	11: IF (OP90_Camera_Trigger AND (NOT OP90_Camera_Done)) OR OP90_Miss_Trigger THEN
			OP90_LH_Camera_Trigger:=1;
			OP90_RH_Camera_Trigger:=1;
			Conv_Cam_Step		  :=15;	
		END_IF

	15:	IF LH_Cam_Completed AND RH_Cam_Completed THEN// (NOT OP90_LH_Camera_Trigger) AND (NOT OP90_RH_Camera_Trigger) THEN //(Temp_Counter_LH<OP90_Camera_FB.OP90_LH_Acquisition_ID AND Temp_Counter_RH<OP90_Camera_FB.OP90_RH_Acquisition_ID )THEN
			OP90_LH_Camera_Trigger:=0;
			OP90_RH_Camera_Trigger:=0;
			OP90_Camera_Trigger :=0;
			OP90_Miss_Trigger	:=0;
			Conv_Cam_Step:=25;
		END_IF  
	   
	25: IF OP90_Camera_FB.OP90_LH_Cam_Result[0]=1 AND OP90_Camera_FB.OP90_RH_Cam_Result[0]=1 THEN
			OP90_LH_Camera_OK:=1;
			OP90_RH_Camera_OK:=1;
			Conv_Cam_Step    :=50;
		ELSIF (OP90_Camera_FB.OP90_LH_Cam_Result[2]<>1 OR OP90_Camera_FB.OP90_RH_Cam_Result[2]<>1) THEN
			OP90_One_Cycle	 :=1;
			Comp_Not_present_Counter:=Comp_Not_present_Counter+1;
			Conv_Cam_Step    :=50;
		ELSIF (OP90_Camera_FB.OP90_LH_Cam_Result[1]=1 OR OP90_Camera_FB.OP90_RH_Cam_Result[1]=1) THEN //AND ( OP90_Camera_FB.OP90_LH_Cam_Result[2]=1 AND OP90_Camera_FB.OP90_RH_Cam_Result[2]=1) THEN			
			IF OP90_Camera_FB.OP90_LH_Cam_Result[0]=1 THEN
				OP90_LH_Camera_OK:=1;
			END_IF
			IF OP90_Camera_FB.OP90_RH_Cam_Result[0]=1 THEN
				OP90_RH_Camera_OK:=1;
			END_IF
			Conv_Cam_Step:=30;
		END_IF	
			
   30: 	IF OP90_Camera_FB.OP90_LH_Cam_Result[1]=1 THEN
	   		OP90_LH_Camera_NOK:=1;
  	    END_IF
		IF OP90_Camera_FB.OP90_RH_Cam_Result[1]=1 THEN
	   		OP90_RH_Camera_NOK:=1;
  	    END_IF
		Conv_Cam_Step:=50;
		
   50:  OP90_Camera_Done:=1;
   		Comp_Not_present_Counter:=0;
   		Temp_Counter_LH:=OP90_Camera_FB.OP90_LH_Acquisition_ID;
		Temp_Counter_RH:=OP90_Camera_FB.OP90_RH_Acquisition_ID;
		IF Camera_Trigger_Ack_OP90 THEN
			Conv_Cam_Step   :=10;
			OP90_Camera_Done:=0;
		END_IF
   	    
END_CASE

END_PROGRAM

// ---- FB/Servo_Conveyor_FB_OP90.TcPOU
FUNCTION_BLOCK Servo_Conveyor_FB_OP90
VAR_INPUT
	Conveyor_Prgrm_Start			: BOOL;
	Conveyor_Prgrm_Reset			: BOOL;
	Conveyor_Continuous_Run			: BOOL;	
	Camera_Trigger_OK				: BOOL;	
	Conveyor_Bypass					: BOOL;
	Fwd_Time_IP						: INT;
	Rev_Time_IP						: INT;
	Conveyor_FWD_Speed				: REAL;
	Conveyor_REV_Speed				: REAL;
	Conveyor_FWD_Position			: REAL;
	Conveyor_REV_Position			: REAL;	
	Velocity_mode					: BOOL;
	LH_Work_Sensor					: BOOL;
	LH_Home_Sensor					: BOOL;
	RH_Work_Sensor					: BOOL;
	RH_Home_Sensor					: BOOL;	
	LH_Camera_OK					: BOOL;
	LH_Camera_NOK					: BOOL;	
	RH_Camera_OK					: BOOL;
	RH_Camera_NOK					: BOOL;
	Track_Overflow					: BOOL;
	//Track_Sensor_FB					: BOOL;
END_VAR
VAR_OUTPUT
	Camera_Trigger_ACK				: BOOL;	
	LH_Work_Coil					: BOOL;
	LH_Home_Coil					: BOOL;
	RH_Work_Coil					: BOOL;
	RH_Home_Coil					: BOOL;	
	Ready_to_Pick					: BOOL;
	Drum_ON							: BOOL;
	Step_Num						: INT;
END_VAR
VAR_IN_OUT
	Camera_trigger						: BOOL;
	One_Cycle							: BOOL;
	Pick_Done						    : BOOL;
	Track_Sensor_FB					    : BOOL;
	Conveyor_Servo_Control_Structure	:  Servo_Control;
END_VAR
VAR
	Conveyor_Speed  : REAL;
	Cyl_Delay 		: TON;
	Cyl_Temp 		: BOOL;
	temp_3			: BOOL;
	cam_ok 			: BOOL;
	con_step_no 	: INT;	
	t1				: ton;
	t2				: ton;
	t3				: ton;
	t4				: ton;	
	count_nok   	: INT;
	forward			: BOOL;
	reverse			: BOOL;
	fwd_time		: INT;
	rev_time		: INT;
	temp            : BOOL;
	VeloCity_Frwd   : REAL := 200;
	Track_Count		: TON;
	Temp_1 : R_TRIG;
	Temp_Cont : BOOL;
	Conti_run : TON;
END_VAR

IF NOT Conveyor_Prgrm_Start OR Conveyor_Servo_Control_Structure.Axis_Error THEN
	con_step_no:=10;
	Camera_Trigger_ACK:=0;
	Ready_to_Pick:=FALSE;
	Conveyor_Servo_Control_Structure.VELmove_Start:=FALSE;
END_IF

IF Conveyor_Bypass THEN
	con_step_no:=10;
	Ready_to_Pick:=1;
	IF Pick_Done THEN
		Pick_Done:=0;
		Ready_to_Pick:=0;
	END_IF
END_IF

IF forward THEN
	Conveyor_Speed:=Conveyor_FWD_Speed;
END_IF
IF reverse THEN
	Conveyor_Speed:=Conveyor_REV_Speed;
END_IF

Conti_run(IN:=(con_step_no=25),PT:=T#2S);

CASE con_step_no OF
		10: IF Conveyor_Prgrm_Start THEN
				con_step_no:=15;
			END_IF
			
		15: LH_Home_Coil:=1;
			RH_Home_Coil:=1;	
			IF LH_Home_Sensor AND RH_Home_Sensor THEN
				LH_Home_Coil:=0;
				RH_Home_Coil:=0;
				con_step_no:= 70;
			END_IF
		
        20:	Ready_to_Pick :=FALSE;
			Pick_Done:= FALSE;
			Conveyor_Servo_Control_Structure.Velocity:= VeloCity_Frwd;		
			Conveyor_Servo_Control_Structure.VELmove_Start:=FALSE;
			IF NOT Conveyor_Servo_Control_Structure.VELmove_Start THEN
				con_step_no:= 25;
			END_IF	
			
		25:	Drum_ON:=1;
			Conveyor_Servo_Control_Structure.VELmove_Start:=TRUE;	
			IF Track_Sensor_FB THEN
				Conveyor_Servo_Control_Structure.VELmove_Start:=FALSE;
				Drum_ON	   :=FALSE;
				con_step_no:= 80;
			END_IF
	
		70: IF NOT Conveyor_Servo_Control_Structure.VELmove_Start THEN
			  Camera_trigger :=TRUE;
			  con_step_no	 := 75;
			END_IF	
					
		75:	IF Camera_Trigger_OK AND NOT Conveyor_Servo_Control_Structure.VELmove_Start AND Conveyor_Servo_Control_Structure.Axis_ready THEN
				IF LH_Camera_OK AND RH_Camera_OK THEN
				 con_step_no:= 100;
				 Camera_Trigger_ACK:=1;
				 fwd_time:=Fwd_Time_IP;
				 count_nok:=0;	
				ELSIF (LH_Camera_NOK) OR (RH_Camera_NOK) AND count_nok<5 THEN
				 count_nok := count_nok +1;
				 con_step_no:= 76;	
				ELSIF count_nok>=5 THEN
	             fwd_time:=3000;
				 con_step_no:= 80; 
				END_IF
			END_IF	
			
		76:	IF LH_Camera_NOK AND NOT Conveyor_Servo_Control_Structure.VELmove_Start THEN
				IF LH_Home_Sensor THEN
					LH_Work_Coil:=TRUE;
					Cyl_Temp:=1;
				END_IF	
				IF Cyl_Delay.Q THEN
					con_step_no:= 77;
				END_IF	
			ELSIF LH_Camera_OK AND RH_Camera_NOK THEN
				con_step_no:= 78;
			END_IF	
			
			
		77: 	IF  LH_Work_Sensor THEN
					LH_Work_Coil:=0;
					LH_Home_Coil:=1;
				END_IF	
				IF LH_Home_Sensor AND NOT LH_Work_Coil AND count_nok<5 THEN
					LH_Home_Coil:=0;
					fwd_time:=Fwd_Time_IP;
				    con_step_no:= 80;
				END_IF
                IF  LH_Home_Sensor AND NOT LH_Work_Coil AND count_nok>=5 THEN
					LH_Home_Coil:=0;
					fwd_time:=3000;
					count_nok:=0;
					//Camera_Trigger_ACK:=1;
				    con_step_no:= 80;	
				END_IF

		78:	IF RH_Camera_NOK AND NOT Conveyor_Servo_Control_Structure.VELmove_Start THEN	
				IF RH_Home_Sensor THEN
					RH_Work_Coil:=TRUE;
					Cyl_Temp:=1;
				END_IF	
				IF Cyl_Delay.Q THEN
					con_step_no:= 79;
				END_IF				
			END_IF		
			
		79: 	IF RH_Work_Sensor THEN
					RH_Work_Coil:=0;
					RH_Home_Coil:=1;				
				END_IF
				IF RH_Home_Sensor AND NOT RH_Work_Coil AND count_nok<5 THEN
					RH_Home_Coil:=0;					
					fwd_time:=Fwd_Time_IP;
				    con_step_no:= 80;
				END_IF
				IF RH_Home_Sensor AND NOT RH_Work_Coil AND count_nok>=5 THEN
					fwd_time:=3000;
					count_nok:=0;
					RH_Home_Coil:=0;
				    con_step_no:= 80;	
				END_IF
			
		80: 	IF Velocity_mode THEN
					IF fwd_time=3000 THEN
			       		count_nok:=0;	
					END_IF
                	Conveyor_Servo_Control_Structure.Velocity:= Conveyor_Speed;				
					forward:=TRUE;
					Conveyor_Servo_Control_Structure.VELmove_Start:=TRUE;	
					IF t2.Q THEN
    					forward:=FALSE;
						Conveyor_Servo_Control_Structure.VELmove_Start:=FALSE;
						Camera_Trigger_ACK:=1;
						con_step_no:= 90;
					END_IF
				ELSE
					Conveyor_Servo_Control_Structure.Velocity:=Conveyor_FWD_Speed;
					Conveyor_Servo_Control_Structure.Position:=Conveyor_FWD_Position;
					Conveyor_Servo_Control_Structure.RELmove_Start:=1;
					Camera_Trigger_ACK:=1;
					con_step_no:= 85;
				END_IF	
				
		85 : 	IF NOT Conveyor_Servo_Control_Structure.RELmove_Start THEN 
					con_step_no:= 90;
				END_IF	
		
		90: IF Velocity_mode THEN
				Conveyor_Servo_Control_Structure.Velocity:= Conveyor_Speed;
				reverse:=TRUE;
				Conveyor_Servo_Control_Structure.VELmove_Start:=TRUE;
				IF t3.Q THEN
 					reverse:=FALSE;
					Conveyor_Servo_Control_Structure.VELmove_Start:=FALSE;
					Camera_Trigger_ACK:=0;
					IF NOT Camera_Trigger_ACK THEN
						con_step_no:= 70;
					END_IF	
				END_IF
			ELSE
				Conveyor_Servo_Control_Structure.Velocity:=ABS(Conveyor_REV_Speed);
				Conveyor_Servo_Control_Structure.Position:=(-Conveyor_REV_Position);
				Conveyor_Servo_Control_Structure.RELmove_Start:=1;
				Camera_Trigger_ACK:=0;
					IF NOT Camera_Trigger_ACK THEN
						con_step_no:= 92;
					END_IF
			END_IF
			
			
		92 : 	IF NOT Conveyor_Servo_Control_Structure.RELmove_Start THEN 
					con_step_no:= 70;
				END_IF
				
		100: IF NOT Conveyor_Servo_Control_Structure.VELmove_Start THEN
				// Camera_Trigger_ACK:=1;
				 Ready_to_Pick:=TRUE;
			 END_IF	
			 IF Pick_Done OR Conveyor_Continuous_Run THEN
				 Ready_to_Pick :=FALSE;
				 Pick_Done:= FALSE;
				 con_step_no:= 80;
			 END_IF	

		101: IF LH_Home_Sensor AND RH_Home_Sensor THEN
					LH_Work_Coil:=TRUE;
					RH_Work_Coil:=TRUE;
					Cyl_Temp:=1;
				END_IF	
				IF Cyl_Delay.Q THEN
					con_step_no:= 102;
				END_IF	

		102: IF RH_Work_Sensor AND LH_Work_Sensor THEN
					RH_Work_Coil:=0;
					LH_Work_Coil:=0;
					RH_Home_Coil:=1;
					LH_Home_Coil:=1;				
				END_IF
				IF RH_Home_Sensor AND LH_Home_Sensor AND NOT RH_Work_Coil AND NOT LH_Work_Coil AND count_nok<5 THEN
					RH_Home_Coil:=0;	
					LH_Home_Coil:=0;				
					fwd_time:=Fwd_Time_IP;
				    con_step_no:= 80;
				END_IF	
				IF RH_Home_Sensor AND LH_Home_Sensor AND NOT RH_Work_Coil AND NOT LH_Work_Coil AND count_nok>=5 THEN
					RH_Home_Coil:=0;	
					LH_Home_Coil:=0;				
					fwd_time:=3000;
				    con_step_no:= 80;
				END_IF		
END_CASE


(*IF Track_Sensor_FB AND NOT Conveyor_Servo_Control_Structure.VELmove_Start THEN
	con_step_no:= 20;
	Track_Sensor_FB:=0;
END_IF*)

Step_Num:=con_step_no;
	
Temp_1(CLK:=Track_Count.Q );
temp:=1;
rev_time:=Rev_Time_IP;

t2(IN:=forward ,PT:=INT_TO_TIME(fwd_time));
t3(IN:=reverse ,PT:=INT_TO_TIME(rev_time));

Cyl_Delay(IN:=Cyl_Temp,PT:=T#600MS);
IF Cyl_Delay.Q THEN
	Cyl_Temp:=0;
END_IF

IF One_Cycle THEN
	con_step_no := 80;
	One_Cycle	:=0;
END_IF

END_FUNCTION_BLOCK

// ---- POUs/Programs/OP110/OP110_MAIN.TcPOU
PROGRAM OP110_MAIN
VAR
	OP110_Modeselection_FB: Mode_Selection_Block1;
	
//	OP110_Cycle_Time: Cycle_Time_FB;
	TP_100ms: TP;
	Pulse_100ms: BOOL;
	Times: LREAL;
	Start: BOOL;
	Gen_Timer: TON;
END_VAR

// Function Calling

OP110_Manual();
OP110_AUTOSEQUENCE();
OP110_Error();
OP110_Initialization_Seq();

//MOdeselection From HMI

IF (OP110_GVL.OP110_HMI_AutoMode AND NOT OP110_GVL.OP110_HMI_ManualMOde AND NOT OP110_GVL.OP110_HMI_StepMode) THEN
	OP110_Modeselection_FB.ModeWord:=1;
	ELSIF (NOT OP110_GVL.OP110_HMI_AutoMode AND OP110_GVL.OP110_HMI_ManualMOde AND NOT OP110_GVL.OP110_HMI_StepMode) THEN
		OP110_Modeselection_FB.ModeWord:=2;
	ELSIF  (NOT OP110_GVL.OP110_HMI_AutoMode AND NOT OP110_GVL.OP110_HMI_ManualMOde AND  OP110_GVL.OP110_HMI_StepMode) THEN
		OP110_Modeselection_FB.ModeWord:=3;
    ELSE   
		OP110_Modeselection_FB.ModeWord:=0;
END_IF
	
OP110_Modeselection_FB(
	ModeWord:= , 
	HomeConditionOK:=OP110_HomeConditionOK , 
	OperationEnable:=OP110_AutoSelected, 
	StartPB:=OP110_HMI_CycleStart , 
	SafetyAndNOError:= OP110_Safety_OK, 
	ModeAck:=TRUE, 
	HomingINProgress:=OP110_HomeRunning , 
	TempHomeOK:=OP110_Temp_hmeOK , 
	ResetPB:= , 
	AutoSelected=> OP110_AutoSelected, 
	ManualSelected=> OP110_ManualSelected, 
	StepSelected=>OP110_StepSelected , 
	ModeSelAck_Indication=> , 
	StatusDisplay=> , 
	AutoRunning:=OP110_AutoRunning, 
	StepRunning:=OP110_StepRunning , 
	StartEnable:=OP110_StartEnable  , 
	MachineStop:=OP110_Machine_Stop );

//IF OP110_AutoSelected OR OP110_ManualSelected THEN
//	SR110_Vert_servo.bEnable:=TRUE;
//END_IF
OP110_Safety_OK:=OperationEnable;

IF NOT SR110_Vert_servo.bAxisHomed THEN
	SR110_Vert_servo_not_Home:=TRUE;
ELSE
	SR110_Vert_servo_not_Home:=FALSE;
END_IF

IF OP110_GVL.SR110_Vert_servo.bAxisError  THEN
	OP110_ErrorActive:=TRUE;
END_IF

IF OP110_Stop_Request AND NOT OP110_STN_ENABLE THEN
	OP110_Machine_Stop:=1;
END_IF
Gen_Timer(IN:=OP110_Machine_Stop,PT:=T#5S);
IF Gen_Timer.Q THEN
	OP110_Machine_Stop:=0;
END_IF

END_PROGRAM

// ---- POUs/Programs/OP110/OP110_MANUAL.TcPOU
PROGRAM OP110_MANUAL
VAR

//	SR20_Vert_servo_ctrl:Servo_Control_1;
	SR110_Vert_servo_Axis :AXIS_REF;

	OP110_LH_OIL_SPIN_M: BOOL;
	OP110_RH_OIL_SPIN_M: BOOL;
	OP110_LH_OIL_SPRAY_M: BOOL;
	OP110_RH_OIL_SPRAY_M: BOOL;
	temp_safe: BOOL;
	temp:BOOL;
	temp_1: BOOL;
	Op110Enable: BOOL;
END_VAR

IF ( MANUAL_SELECTED OR OP110_HMI_ManualMode )AND NOT ERROR_ACTIVE THEN
  
    IF OP110_LH_OIL_SPIN_M THEN
	    O110_LH_OIL_SPIN_ON_Q1260_1:=TRUE;
	ELSE 
		O110_LH_OIL_SPIN_ON_Q1260_1:=FALSE;
	END_IF
	
    IF OP110_RH_OIL_SPIN_M THEN
	    O110_RH_OIL_SPIN_ON_Q1260_3:=TRUE;
	ELSE 
		O110_RH_OIL_SPIN_ON_Q1260_3:=FALSE;
	END_IF	  
	
	IF OP110_LH_OIL_SPRAY_M THEN
	   O110_LH_OIL_DISPN_ON_Q1260_0:=TRUE;
	   O110_LH_OIL_DISPN_FRL_VLVE_ON_Q401_6:=1;
	ELSE 
	   O110_LH_OIL_DISPN_ON_Q1260_0:=FALSE;
	   O110_LH_OIL_DISPN_FRL_VLVE_ON_Q401_6:=0;
	END_IF
	
	IF OP110_RH_OIL_SPRAY_M THEN
	   O110_RH_OIL_DISPN_ON_Q1260_2:=TRUE;
	   O110_RH_OIL_DISPN_FRL_VLVE_ON_Q401_4 := 1;
	ELSE 
	   O110_RH_OIL_DISPN_ON_Q1260_2:=FALSE;
	   O110_RH_OIL_DISPN_FRL_VLVE_ON_Q401_4 :=0;
	END_IF	
	
END_IF

OP110_VERT_SERVO_POSITION := SR20_Vert_servo.Actual_position;
//SR20_Vert_servo_ctrl.ABSmove_Start := OP110_VERT_SERVO_STRT;
OP110_SERVO_POS_DONE	:= SR20_Vert_servo.bABS_Pos_done ;
//SR20_Vert_servo.fTargetPosition := OP110_VERT_SERVO_TARGET;

IF In_Range(SR110_Vert_servo_status.actualPosition,OP110_VERT_SERVO_SFE_WRK_POS,1) THEN
	OP110_SERVO_ON_SFE_WRK := TRUE;
ELSE
	OP110_SERVO_ON_SFE_WRK := FALSE;
END_IF

IF In_Range(SR110_Vert_servo_status.actualPosition,OP110_VERT_SERVO_HME_POS,1) THEN
	OP110_SERVO_ON_HOME := TRUE;
ELSE
	OP110_SERVO_ON_HOME := FALSE;
END_IF

IF In_Range(SR110_Vert_servo_status.actualPosition,OP110_VERT_SERVO_WRK_POS,2) THEN
	OP110_SERVO_ON_WRK := TRUE;
ELSE
	OP110_SERVO_ON_WRK := FALSE;
END_IF		

OP110_VERT_SERVO_SFE_WRK_POS := OP110_HMI_Safe_Work;
OP110_VERT_SERVO_HME_POS     := OP110_HMI_Safe_Home;
OP110_VERT_SERVO_WRK_POS     := OP110_VERT_SERVO_WORK_POS;

//SR20_Vert_servo_status.jogPos:=OP110_HMI_Jog_Pos;
//SR20_Vert_servo_status.jogNeg:=OP110_HMI_Jog_Neg;
	
OP110_GVL.SR110_Vert_servo(
	bAxis1_Ref_Switch:= temp, 
	bInit:= , 
	bErrorReset:=OP110_Servo_Reset OR Servo_Reset , 
	bEnable:=Servo_Enable, 
	bMoveVelocity:= , 
	bHalt:= , 
	bManualMode:= OP110_ManualSelected AND MANUAL_SELECTED,
	fHomePos:= , 
	fOverride:= , 
	fTargetPosition:=SR110_Vert_servo_ctrl.Position , 
	fTargetVelocity:=SR110_Vert_servo_ctrl.Velocity , 
	fAcc:= , 
	fDec:= ,
	Servo_High_Limit:= OP110_HMI_High_Limit,	
	Servo_Low_Limit:=  OP110_HMI_Low_Limit,	 
	bmove_home:=SR110_Vert_servo_ctrl.Axis_Home_Cmd ,
	baxis_in_home_pos=>SR110_Vert_servo_ctrl.Axis_In_Home ,
	Safe_move_Conditions:=Servo_Safety,
	Axis:= SR110_Vert_servo_Axis , 
	HME_WRITE_ADD:= 16#500E,	
	bHome:=SR110_Vert_servo_ctrl.Bsethome , 
    bSetPosition:=SR110_Vert_servo_ctrl.Bsetpos , 
	bMoveAbsolute:=SR110_Vert_servo_ctrl.ABSmove_Start , 
	bMoveRelative:=SR110_Vert_servo_ctrl.RELmove_Start ,
	bMoveTorque :=SR110_Vert_servo_ctrl.Torque_mode_Start, 
	stManualModeAxis:=SR110_Vert_servo_status , 
	sAxisState=>SR110_Vert_servo_ctrl.Axis_State , 
	bAxis_ready=>SR110_Vert_servo_ctrl.Axis_ready , 
	bAxisInPosition=> SR110_Vert_servo_ctrl.Axis_In_Pos, 
	bAxisError=>SR110_Vert_servo_ctrl.Axis_Error , 
	bAxisEnabled=> SR110_Vert_servo_ctrl.Axis_Enabled, 
	bAxisHomed=> SR110_Vert_servo_ctrl.Axis_reference, 
	bSetPositionDone=>   ,
	bsafe_to_move=> ,
	bABS_Pos_done=> SR110_Vert_servo_ctrl.pos_done , 
	bHaltDone=> , 
	bSTOPDone=> , 
	bHomeDone=> , 
	bDone=> );	
	
IF MANUAL_SELECTED THEN
	SR110_Vert_servo_status.targetVelocity:=50;
END_IF

END_PROGRAM

// ---- POUs/Programs/OP110/OP110_AUTOSEQUENCE.TcPOU
PROGRAM OP110_AUTOSEQUENCE
VAR	
//BOOL
	OP110_STN_ERR					: BOOL;
	OP110_LH_A_OIL_Dispense			: BOOL;
	OP110_RH_A_OIL_Dispense			: BOOL;
	OP110_RH_A_OIL_SPIN 				: BOOL;
	OP110_LH_A_OIL_SPIN				: BOOL;
	OP110_LH_OIL_DONE				: BOOL;
	OP110_RH_OIL_DONE				: BOOL;
	OP110_Oil_Range					: BOOL;
//TON
	OP110_Oiling_Timer: TON;
	OP110_Oiling_Pos: REAL :=6;
	check: BOOL;
	OP110_STN_MOVER: INT;
	OP110_WRK_DELAY : TON;
	WRK_DELAY	: INT :=500;
	OP110_Cycle_Time_FB : FB_Cycletime;		
	MOVER_POS_RECHED_R: R_TRIG;
	Dry_Run: BOOL;

END_VAR

IF OP110_AutoSelected AND NOT OP110_ErrorActive AND OperationEnable THEN
	O110_LH_OIL_DISPN_ON_Q1260_0:=TRUE ;
	O110_RH_OIL_DISPN_ON_Q1260_2:=TRUE ;
	O110_LH_OIL_DISPN_FRL_VLVE_ON_Q401_6:=OP110_LH_A_OIL_Dispense;
	O110_RH_OIL_DISPN_FRL_VLVE_ON_Q401_4:=OP110_RH_A_OIL_Dispense;
	O110_LH_OIL_SPIN_ON_Q1260_1:=OP110_RH_A_OIL_SPIN ;
	O110_RH_OIL_SPIN_ON_Q1260_3:=OP110_LH_A_OIL_SPIN;		
END_IF

OP110_OIL_TIMER:=OP110_DLY_OIL_ON;

// AUTO MODE
IF (NOT OP110_AutoSelected OR OP110_ErrorActive OR OP110_HomeRunning OR NOT  OperationEnable ) THEN
	OP110_AutoRunning:= FALSE;
	OP110_AutoSeq:= 10;
	OP110_STN_ENABLE:=FALSE;
	OP110_STN_RUNNING:=FALSE;
END_IF	

IF ( OP110_ErrorActive OR OP110_HomeRunning OR NOT OperationEnable ) THEN
	O110_LH_OIL_DISPN_ON_Q1260_0 :=0;
	O110_RH_OIL_DISPN_ON_Q1260_2 :=0;
	O110_LH_OIL_SPIN_ON_Q1260_1  :=0;
	O110_RH_OIL_SPIN_ON_Q1260_3  :=0;
END_IF
																									
CASE OP110_AutoSeq OF
		
		10: IF (OP110_AutoSelected) THEN		// Check Automode Selected
				OP110_AutoSeq:=20;
	        END_IF
		
	    20:IF ( NOT OP110_ErrorActive) THEN		//Check No error
		       OP110_AutoSeq:=30;
      	   END_IF
		   
      	30:IF (NOT OP110_HomeRunning) THEN		//Check No Homerunning
      		   OP110_AutoSeq :=40;
      	   END_IF
		   
        40:IF (OP110_Main.OP110_Modeselection_FB.TempHomeOK)THEN	//Check Machine in Home
      		   OP110_AutoSeq:= 50;
      	   END_IF
		   
      	50:IF ( OP110_STN_ENABLE AND OP110_STN_RUNNING ) THEN		// Check Operation Completed Reset
      		   OP110_AutoSeq:=70;
		   ELSE
	   		   OP110_AutoSeq:=60;
      	   END_IF
	   60:IF  ( AUTO_RUNNING OR (NOT AUTO_RUNNING AND OP110_HMI_CycleStart )) THEN		//Machine Start in Fully Automatic or Press Cycle Start For Semi Automatic
		    OP110_HomeConditionOK:=TRUE;
	 			IF( OP110_Main.OP110_Modeselection_FB.HomeConditionOK AND OP110_AutoSelected) THEN
					OP110_AutoRunning:=TRUE;
					OP110_StepRunning:= FALSE;
				
				ELSIF (OP110_Main.OP110_Modeselection_FB.HomeConditionOK AND OP110_StepSelected) THEN
					OP110_AutoRunning:=FALSE;
					OP110_StepRunning:= TRUE;
				END_IF;
		  END_IF
		   IF ((OP110_AutoRunning OR OP110_StepRunning) AND OP110_StartEnable) THEN
				OP110_AutoSeq:= 70;
		   END_IF

      	70:  // SERVO POSITION SAFE CHECK
	       IF (OP110_SERVO_ON_SFE_WRK OR OP110_SERVO_ON_HOME)AND OP110_SERVO_POS_DONE AND NOT SR110_Vert_servo_ctrl.ABSmove_Start THEN 
	         SR110_Vert_servo_ctrl.Position := OP110_VERT_SERVO_WRK_POS;
			 SR110_Vert_servo_ctrl.Velocity := OP110_HMI_Servo_Speed;
			 IF SR110_Vert_servo_ctrl.Position=OP110_VERT_SERVO_WRK_POS THEN
 				OP110_AutoSeq:=75;
			 END_IF	
	       END_IF
			   
		75: // WAITING FOR MOVER AND MOVING SERVO TO TARGET POSITION
			IF OP110_STN_ENABLE THEN
			 SR110_Vert_servo_ctrl.ABSmove_Start:=TRUE;
			 OP110_STN_RUNNING :=1;
			 OP110_LH_OIL_OK:=FALSE;
			 OP110_RH_OIL_OK:=FALSE;			 
			 OP110_AutoSeq:=80;
			END_IF
			
		80: // START THE SPINNER OK COMPONENT FIXTURE
			 IF OP110_FIXTURE_1=90 AND OP110_FIXTURE_2<>90  THEN
			   OP110_LH_A_OIL_Dispense:=1;
			   OP110_AutoSeq:=100;			   
			 ELSIF OP110_FIXTURE_2=90 AND OP110_FIXTURE_1<>90 THEN
			   OP110_RH_A_OIL_Dispense:=1;
			   OP110_AutoSeq:=100;			   
			 ELSIF OP110_FIXTURE_1=90 AND OP110_FIXTURE_2=90 THEN  
				OP110_LH_A_OIL_Dispense:=1;
				OP110_RH_A_OIL_Dispense:=1;
			    OP110_AutoSeq:=100;				
			 ELSIF OP110_FIXTURE_1<>90 AND OP110_FIXTURE_2<>90 AND OP110_SERVO_ON_WRK THEN
			 	OP110_AutoSeq:=120;	
			 END_IF	
	
		100: IF OP110_WRK_DELAY.Q  THEN
				OP110_RH_A_OIL_SPIN:=1;
		        OP110_LH_A_OIL_SPIN:=1;
				SR110_Vert_servo_ctrl.Position:=(OP110_VERT_SERVO_WRK_POS-OP110_Oil_Position_Offset);
				SR110_Vert_servo_ctrl.Velocity:=OP110_Oiling_Velocity;
				OP110_AutoSeq:=110;
			 END_IF
			 OP110_CURR_MOVER			:= OP110_STN_MOVER;
			 
		110: SR110_Vert_servo_ctrl.ABSmove_Start:=TRUE;	
			 OP110_AutoSeq:=115;
			
		115: IF In_Range(SR110_Vert_servo_status.actualPosition,(OP110_VERT_SERVO_WRK_POS-OP110_Oil_Position_Offset),1) AND NOT SR110_Vert_servo_ctrl.ABSmove_Start THEN
				OP110_LH_OIL_OK:=1;
				OP110_RH_OIL_OK:=1;
				OP110_RH_A_OIL_SPIN:=0;
		        OP110_LH_A_OIL_SPIN:=0;	
				OP110_LH_A_OIL_Dispense:=0;
				OP110_RH_A_OIL_Dispense:=0;			
				OP110_AutoSeq:=120;
			 END_IF
		      		
		120:SR110_Vert_servo_ctrl.Position :=OP110_VERT_SERVO_SFE_WRK_POS;
			SR110_Vert_servo_ctrl.Velocity := OP110_HMI_Servo_Speed;
			IF OP110_LH_OIL_OK THEN
				MOVER_CMP_STATUS[OP110_CURR_MOVER][1]	:=110;
			ELSE
				MOVER_CMP_STATUS[OP110_CURR_MOVER][1]	:=110;				
			END_IF
			IF OP110_RH_OIL_OK THEN
				MOVER_CMP_STATUS[OP110_CURR_MOVER][2]	:=110;
			ELSE                                 
				MOVER_CMP_STATUS[OP110_CURR_MOVER][2]	:=110;				
			END_IF	
			OP110_AutoSeq:=140;				  		
			
		140:  IF NOT SR110_Vert_servo_ctrl.ABSmove_Start THEN			 
			   SR110_Vert_servo_ctrl.ABSmove_Start:=TRUE;
			   OP110_AutoSeq:=160;
			 END_IF				  
	     	  	  	
		160: // SERVO DONE AND RESET THE DONE BITS
			IF NOT SR110_Vert_servo_ctrl.ABSmove_Start AND OP110_SERVO_ON_SFE_WRK THEN
			  SR110_Vert_servo_ctrl.ABSmove_Start:=FALSE;
			  OP110_STN_RUNNING  :=0;
			  OP110_STN_ENABLE:=FALSE;
			  OP110_RH_A_OIL_SPIN:=0;
			  OP110_LH_A_OIL_SPIN:=0;
			 STATION_DONE[OP110_CURR_MOVER][OP110_XTS_POS_NO]			:= TRUE;
			  OP110_AutoSeq:=70;			
			END_IF

END_CASE

OP110_Cycle_Time_FB(i_b_startTime:=OP110_STN_ENABLE , i_b_stopTime:= NOT OP110_STN_ENABLE , o_t_StationTime=>OP110_Cycle_time );					

OP110_WRK_DELAY(IN:=OP110_SERVO_ON_WRK,PT:=INT_TO_TIME(WRK_DELAY));

Dry_Run:=All_Station_Dry_Run;
IF Dry_Run THEN
	OP110_FIXTURE_1:=90;
	OP110_FIXTURE_2:=90;
ELSE 
	OP110_FIXTURE_1:=MOVER_CMP_STATUS[OP110_STN_MOVER][1];
	OP110_FIXTURE_2:=MOVER_CMP_STATUS[OP110_STN_MOVER][2];	
END_IF	
//Timers
//OP110_Oiling_Timer(IN:=OP110_LH_A_OIL_Dispense OR OP110_RH_A_OIL_Dispense, PT:=INT_TO_TIME(OP110_OIL_TIMER) , Q=> , ET=> );
//IF OP110_Oiling_Timer.Q THEN
//	OP110_LH_A_OIL_Dispense:=0;
//	OP110_RH_A_OIL_Dispense:=0;
//END_IF				


//############################		OP110 STATION ENABLE CONDITION		##########################

	OP110_STN_MOVER					:= MOVER_POSITION[OP110_XTS_POS_NO];
	IF AUTO_WITH_XTS THEN
	IF OP110_STN_MOVER>0 THEN		
	IF NOT(END_OF_CYCLE AND MOVER_CMP_STATUS[OP110_STN_MOVER][1]=5 AND MOVER_CMP_STATUS[OP110_STN_MOVER][2]=5)THEN
		OP110_STN_ENABLE			:= MOVER_POS_RECHED[OP110_STN_MOVER] AND ((MOVER_CMP_STATUS[OP110_STN_MOVER][1]=90)OR
										(MOVER_CMP_STATUS[OP110_STN_MOVER][2]=90))AND STATION_ENABLE_CONTROL;
	
	ELSE
		STATION_DONE[OP110_STN_MOVER][OP110_XTS_POS_NO]			:= TRUE;		
	END_IF
	ELSE
		OP110_STN_ENABLE			:= FALSE;
	END_IF																			
	END_IF

END_PROGRAM

// ---- POUs/Programs/OP110/OP110_ERROR.TcPOU
PROGRAM OP110_ERROR
VAR
	OP110_StErr_1: TON;
	OP110_Step_Err_2: TON;
	OP110_StepErr_3: TON;
	OP110_StErr_4: TON;
	OP110_Step_Err_5: TON;
	OP110_StepErr_6: TON;
//	end: INT;
END_VAR

//Reset ErrorActive
IF (OP110_HMI_Reset OR Servo_Reset) THEN 
	OP110_GVL.OP110_ErrorActive:= FALSE;
	OP110_GVL.OP110_ErrorWord_0:= 0;
	OP110_GVL.OP110_ErrorWord_1:= 0;
	OP110_GVL.OP110_ErrorWord_2:= 0;	
END_IF

//(OP110_GVL.OP110_ErrorWord_0<>0) OR
// Set ERROR ACTIVE
IF ( (OP110_GVL.OP110_ErrorWord_1<>0) OR (OP110_GVL.OP110_ErrorWord_2<>0)) THEN
	OP110_GVL.OP110_ErrorActive:= TRUE;
END_IF


OP110_ErrorWord_0.0:= SR110_Vert_servo_ctrl.Axis_Error;
OP110_ErrorWord_0.1:= NOT OperationEnable;
// Auto Seq Step Error
//Servo not reaching work position
OP110_StErr_1(IN:=(OP110_GVL.OP110_AUTO_STP_NO=80) , PT:=T#5S , Q=> , ET=> );
IF (OP110_GVL.OP110_AUTO_STP_NO=80 AND NOT OP110_GVL.OP110_SERVO_ON_WRK AND OP110_StErr_1.Q) THEN
	OP110_GVL.OP110_ErrorWord_0.2:=TRUE;
END_IF

// Servo Not Reached home position or safe-work position
OP110_Step_Err_2(IN:=OP110_GVL.OP110_AUTO_STP_NO=160, PT:=T#5S , Q=> , ET=> );
IF (OP110_GVL.OP110_AUTO_STP_NO=160 AND NOT OP110_SERVO_ON_SFE_WRK AND OP110_Step_Err_2.Q) THEN
	OP110_GVL.OP110_ErrorWord_0.3:=TRUE;
END_IF
OP110_GVL.OP110_ErrorWord_0.4:=0;
//OP110_StepErr_3(IN:=( OP110_HomeRunning AND (OP110_Homing_Seq=10) AND NOT SR110_Vert_servo_ctrl.Axis_In_Home), PT:=T#10S , Q=> , ET=> );
//IF OP110_StepErr_3.Q THEN
//	OP110_GVL.OP110_ErrorWord_0.4:=TRUE;
//END_IF

END_PROGRAM

// ---- POUs/Programs/OP110/OP110_Initialization_Seq.TcPOU
PROGRAM OP110_Initialization_Seq
VAR
END_VAR

IF (SR110_Vert_servo_ctrl.Axis_In_Home)THEN
OP110_Temp_hmeOK:=TRUE;
OP110_HomeRunning:=FALSE;
OP110_Homing_Seq:=0;
ELSE
	OP110_Temp_hmeOK:=FALSE;	
END_IF

CASE OP110_Homing_Seq OF
	0: IF (OP110_AutoSelected AND NOT OP110_HomeRunning AND NOT OP110_ErrorActive AND NOT OP110_AutoRunning AND NOT OP110_StepRunning AND NOT OP110_Temp_hmeOK) THEN
		OP110_HomeRunning:=TRUE;
		OP110_Homing_Seq:=10;	
	   END_IF
	10:IF (OP110_HomeRunning AND (OP110_HMI_Homing OR HMI_Reset))THEN 
			IF (SR110_Vert_servo_ctrl.Axis_In_Home) THEN 
				//OP110_Homing_Seq:=110;
				SR110_Vert_servo_ctrl.Axis_Home_Cmd:=FALSE;
			ELSE
				SR110_Vert_servo_ctrl.Position:=0;
				SR110_Vert_servo_ctrl.Velocity:=100;
				SR110_Vert_servo_ctrl.ABSmove_Start:=TRUE;
				SR110_Vert_servo_ctrl.Axis_Home_Cmd:=TRUE;
	    	END_IF
			IF SR110_Vert_servo_ctrl.Axis_In_Home THEN
			  OP110_Homing_Seq:=20;			
			END_IF
	   END_IF		
	20:	OP110_Homing_Seq:=0;
		OP110_HomeRunning:=FALSE;
		OP110_HMI_Homing:=FALSE;
END_CASE

END_PROGRAM

// ---- POUs/Programs/OP120/OP120_Main.TcPOU
PROGRAM OP120_Main
VAR
	OP120_Modeselection_FB: Mode_Selection_Block1;
	

	OP120_Vaccum1_Bit2: BOOL;
	OP120_Vaccum1_Bit6: BOOL;
	OP120_Vaccum1_Bit3: BOOL;
	OP120_Vaccum1_Bit4: BOOL;
	OP120_Vaccum1_Bit5: BOOL;
	OP120_Vaccum1_Bit7: BOOL;
	OP120_Vaccum_Byte2_bit0: BOOL;
	OP120_Vaccum_Byte2_bit1: BOOL;
	OP120_Vaccum_Byte2_bit2: BOOL;
	OP120_Vaccum_Byte2_bit3: BOOL;
	OP120_Vaccum_Byte2_bit4: BOOL;
	OP120_Vaccum_Byte2_bit5: BOOL;
	OP120_Vaccum_Byte2_bit6: BOOL;
	OP120_Vaccum_Byte2_bit7: BOOL;
	OP120_Vaccum2_Bit3: BOOL;
	OP120_Vaccum2_Bit4: BOOL;
	OP120_Vaccum2_Bit2: BOOL;
	OP120_Vaccum2_Bit5: BOOL;
	OP120_Vaccum2_Bit6: BOOL;
	OP120_Vaccum2_Bit7: BOOL;
	OP120_Vaccum2_Byte2_bit0: BOOL;
	OP120_Vaccum2_Byte2_bit1: BOOL;
	OP120_Vaccum2_Byte2_bit2: BOOL;
	OP120_Vaccum2_Byte2_bit3: BOOL;
	OP120_Vaccum2_Byte2_bit4: BOOL;
	OP120_Vaccum2_Byte2_bit5: BOOL;
	OP120_Vaccum2_Byte2_bit6: BOOL;
	OP120_Vaccum2_Byte2_bit7: BOOL;
END_VAR

op120_camera_FB();
OP120_Manual();
Op120_Error();

OP120_Initialization_Seq();
OP120_AutoSequence();
OP120_feed_Conveyor();
OP120_LockInsert_AutoSequence();

OP120_Sing_Auto_PRG();


IF (OP120_HMI_AutoMode AND NOT OP120_HMI_ManualMOde AND NOT OP120_HMI_StepMode) THEN
	OP120_Modeselection_FB.ModeWord:=1;
	ELSIF (NOT OP120_HMI_AutoMode AND OP120_HMI_ManualMOde AND NOT OP120_HMI_StepMode) THEN
		OP120_Modeselection_FB.ModeWord:=2;
	ELSIF  (NOT OP120_HMI_AutoMode AND NOT OP120_HMI_ManualMOde AND  OP120_HMI_StepMode) THEN
		OP120_Modeselection_FB.ModeWord:=3;
    ELSE   
		OP120_Modeselection_FB.ModeWord:=0;
END_IF
	





OP120_Modeselection_FB(
	ModeWord:= , 
	HomeConditionOK:=OP120_HomeCondition_OK , 
	OperationEnable:=OperationEnable , 
	StartPB:= , 
	SafetyAndNOError:=OperationEnable , 
	ModeAck:=TRUE , 
	HomingINProgress:= , 
	TempHomeOK:=OP120_Temp_Home_OK , 
	ResetPB:= , 
	AutoSelected=>OP120_AutoSelected , 
	ManualSelected=>OP120_ManualSelected , 
	StepSelected=>OP120_StepSelected , 
	ModeSelAck_Indication=> , 
	StatusDisplay=> , 
	AutoRunning:=OP120_AutoRunning , 
	StepRunning:=OP120_StepRunning , 
	StartEnable:=OP120_StartEnable , 
	MachineStop:=OP120_Machine_Stop );
	
	IF (OP120_AutoSelected OR  OP120_StepSelected ) THEN
		OP120_GVL.OP120_Auto:=TRUE;
		O120_ROB_MAN_AUTO_MODE_Q709_4:=TRUE;
		//OP120_SI_Dry_Run:=TRUE;
		OP120_Robo_Out6002:=1;
		
		ELSE
			OP120_GVL.OP120_Auto:=FALSE;
			O120_ROB_MAN_AUTO_MODE_Q709_4:=FALSE;
			OP120_Robo_Out6002:=0;
		END_IF
IF OP120_Auto AND NOT OP120_ManualSelected AND NOT OP120_HomeRunning THEN
	OP120_Robo_Out6001:=1;
END_IF
	
	(*OP120_Vaccum1_Bit0:=OP120_Vaccuum_IP_Port5_Byte1.7;
	OP120_Vaccum1_Bit1:=OP120_Vaccuum_IP_Port5_Byte1.6;
	OP120_Vaccum1_Bit2:=OP120_Vaccuum_IP_Port5_Byte1.5;
	OP120_Vaccum1_Bit3:=OP120_Vaccuum_IP_Port5_Byte1.4;
	OP120_Vaccum1_Bit4:=OP120_Vaccuum_IP_Port5_Byte1.3;
	OP120_Vaccum1_Bit5:=OP120_Vaccuum_IP_Port5_Byte1.2;
	OP120_Vaccum1_Bit6:=OP120_Vaccuum_IP_Port5_Byte1.1;
	OP120_Vaccum1_Bit7:=OP120_Vaccuum_IP_Port5_Byte1.0;
	
	OP120_Vaccum_Byte2_bit0:=OP120_Vaccuum_IP_Port5_Byte2.7;
	OP120_Vaccum_Byte2_bit1:=OP120_Vaccuum_IP_Port5_Byte2.6;
	OP120_Vaccum_Byte2_bit2:=OP120_Vaccuum_IP_Port5_Byte2.5;
	OP120_Vaccum_Byte2_bit3:=OP120_Vaccuum_IP_Port5_Byte2.4;
	OP120_Vaccum_Byte2_bit4:=OP120_Vaccuum_IP_Port5_Byte2.3;
	OP120_Vaccum_Byte2_bit5:=OP120_Vaccuum_IP_Port5_Byte2.2;
	OP120_Vaccum_Byte2_bit6:=OP120_Vaccuum_IP_Port5_Byte2.1;*)
	OP120_Vaccum1_Bit0:=OP120_Vaccuum_IP_Port5_Byte2.0;
	
(*OP120_Vaccum2_Bit0:=OP120_Vaccuum_IP_Port6_Byte1.7;
	OP120_Vaccum2_Bit1:=OP120_Vaccuum_IP_Port6_Byte1.6;
	OP120_Vaccum2_Bit2:=OP120_Vaccuum_IP_Port6_Byte1.5;
	OP120_Vaccum2_Bit3:=OP120_Vaccuum_IP_Port6_Byte1.4;
	OP120_Vaccum2_Bit4:=OP120_Vaccuum_IP_Port6_Byte1.3;
	OP120_Vaccum2_Bit5:=OP120_Vaccuum_IP_Port6_Byte1.2;
	OP120_Vaccum2_Bit6:=OP120_Vaccuum_IP_Port6_Byte1.1;
	OP120_Vaccum2_Bit7:=OP120_Vaccuum_IP_Port6_Byte1.0;
	
	OP120_Vaccum2_Byte2_bit0:=OP120_Vaccuum_IP_Port6_Byte2.7;
	OP120_Vaccum2_Byte2_bit1:=OP120_Vaccuum_IP_Port6_Byte2.6;
	OP120_Vaccum2_Byte2_bit2:=OP120_Vaccuum_IP_Port6_Byte2.5;
	OP120_Vaccum2_Byte2_bit3:=OP120_Vaccuum_IP_Port6_Byte2.4;
	OP120_Vaccum2_Byte2_bit4:=OP120_Vaccuum_IP_Port6_Byte2.3;
	OP120_Vaccum2_Byte2_bit5:=OP120_Vaccuum_IP_Port6_Byte2.2;
	OP120_Vaccum2_Byte2_bit6:=OP120_Vaccuum_IP_Port6_Byte2.1;*)
	OP120_Vaccum2_Bit0:=OP120_Vaccuum_IP_Port6_Byte2.0;

END_PROGRAM

// ---- POUs/Programs/OP120/op120_camera_FB.TcPOU
PROGRAM op120_camera_FB
/// op 120 color cam 1
VAR
	op120_color_cam_1 			              : FB_Cognex_ProfiNET_1;
	op120color1_Camera_Trigger		          : BOOL;
	op120color1_Camera_Job_Change_start       : BOOL;
	op120color1_Camera_Error			      : BOOL;
	op120color1_Camera_Ready			      : BOOL;
	op120color1_Camera_Online		          : BOOL;	
	
	op120color1_Acquisition_Status AT %I*      :Acquisition_Status;
	op120color1_Inspection_Status  AT %I*      :Inspection_Status;	
	op120color1_Acquisition_ID     AT %I*      :UINT;
	op120color1_Inspection_ID   	 AT %I*       :UINT;
	op120color1_Error_code      	 AT %I*       :UINT;
	op120color1_Current_Job_ID  	 AT %I*       :UINT;
	op120color1_Result_code     	 AT %I*       :UINT;
	op120color1_Cam_Result      	 AT %I*       :ARRAY[0..63] OF BYTE;

	op120color1_Acquisition_Control AT %Q*     : Acquisition_Control;
	op120color1_Inspection_Control  AT %Q*     : Inspection_Control;
	op120color1_Command_word		  AT %Q*      : UINT;
	Error_status				              : STRING;
	op120color1_Target_Job_ID				  : UINT;
	op120color1_Loaded_Job_ID		    	  : UINT;
	op120color1_Union                          : UNION_64Byte;
	op120color1_Job_Change_Complete		      : BOOL;
	op120color1_Job_Change_Error   		      : BOOL;
	op120color1_Picture_Taken      		      : BOOL;
	
	
	
	
	
	
END_VAR
 /// op 120 color cam 2//
VAR
 op120_color_cam_2                         : FB_Cognex_ProfiNET_1;
 op120color2_Camera_Trigger                 : BOOL;
 op120color2_Camera_Job_Change_start        : BOOL;
 op120color2_Camera_Error                   : BOOL;
 op120color2_Camera_Ready                   : BOOL;
 op120color2_Camera_Online                  : BOOL; 
 
 op120color2_Acquisition_Status AT %I*      :Acquisition_Status;
 op120color2_Inspection_Status  AT %I*      :Inspection_Status; 
 op120color2_Acquisition_ID     AT %I*      :UINT;
 op120color2_Inspection_ID     AT %I*       :UINT;
 op120color2_Error_code        AT %I*       :UINT;
 op120color2_Current_Job_ID    AT %I*       :UINT;
 op120color2_Result_code       AT %I*       :UINT;
 op120color2_Cam_Result        AT %I*       :ARRAY[0..63] OF BYTE;

 op120color2_Acquisition_Control AT %Q*     : Acquisition_Control;
 op120color2_Inspection_Control  AT %Q*     : Inspection_Control;
 op120color2_Command_word    AT %Q*         : UINT;
 Error_status_1                               : STRING;
 op120color2_Target_Job_ID                  : UINT;
 op120color2_Loaded_Job_ID                  : UINT;
 op120color2_Union                          : UNION_64Byte;
 op120color2_Job_Change_Complete            : BOOL;
 op120color2_Job_Change_Error               : BOOL;
 op120color2_Picture_Taken                  : BOOL;


END_VAR

VAR
 op120_orient_cam_1                         : FB_Cognex_ProfiNET_1;
 op120orient1_Camera_Trigger                : BOOL;
 op120orient1_Camera_Job_Change_start       : BOOL;
 op120orient1_Camera_Error                  : BOOL;
 op120orient1_Camera_Ready                  : BOOL;
 op120orient1_Camera_Online                 : BOOL; 
 
 op120orient1_Acquisition_Status AT %I*          :Acquisition_Status;
 op120orient1_Inspection_Status  AT %I*          :Inspection_Status; 
 op120orient1_Acquisition_ID     AT %I*          :UINT;
 op120orient1_Inspection_ID     AT %I*           :UINT;
 op120orient1_Error_code        AT %I*           :UINT;
 op120orient1_Current_Job_ID    AT %I*           :UINT;
 op120orient1_Result_code       AT %I*           :UINT;
 op120orient1_Cam_Result        AT %I*           :ARRAY[0..63] OF BYTE;
 
 op120orient1_User_Data        AT %Q*           :ARRAY[0..63] OF BYTE;
 op120orient1_Acquisition_Control AT %Q*         :Acquisition_Control;
 op120orient1_Inspection_Control  AT %Q*         : Inspection_Control;
 op120orient1_Command_word    AT %Q*          : UINT;
 Error_status_3                  : STRING;
 op120orient1_Target_Job_ID             : UINT;
 op120orient1_Loaded_Job_ID                : UINT;
 op120orient1_Union                              : UNION_64Byte;
 op120orient1_Job_Change_Complete            : BOOL;
 op120orient1_Job_Change_Error               : BOOL;
 op120orient1_Picture_Taken                  : BOOL;
END_VAR


VAR
op120_orient_cam_2                        : FB_Cognex_ProfiNET_1;
 op120orient2_Camera_Trigger                : BOOL;
 op120orient2_Camera_Job_Change_start       : BOOL;
 op120orient2_Camera_Error                  : BOOL;
 op120orient2_Camera_Ready                  : BOOL;
 op120orient2_Camera_Online                 : BOOL; 
 
 op120orient2_Acquisition_Status AT %I*          :Acquisition_Status;
 op120orient2_Inspection_Status  AT %I*          :Inspection_Status; 
 op120orient2_Acquisition_ID     AT %I*          :UINT;
 op120orient2_Inspection_ID     AT %I*           :UINT;
 op120orient2_Error_code        AT %I*           :UINT;
 op120orient2_Current_Job_ID    AT %I*           :UINT;
 op120orient2_Result_code       AT %I*           :UINT;
 op120orient2_Cam_Result        AT %I*           :ARRAY[0..63] OF BYTE;
 
 op120orient2_User_Data        AT %Q*           :ARRAY[0..63] OF BYTE;
 op120orient2_Acquisition_Control AT %Q*         :Acquisition_Control;
 op120orient2_Inspection_Control  AT %Q*         : Inspection_Control;
 op120orient2_Command_word    AT %Q*          : UINT;
 Error_status_2                  : STRING;
 op120orient2_Target_Job_ID             : UINT;
 op120orient2_Loaded_Job_ID                : UINT;
 op120orient2_Union                              : UNION_64Byte;
 op120orient2_Job_Change_Complete            : BOOL;
 op120orient2_Job_Change_Error               : BOOL;
 op120orient2_Picture_Taken                  : BOOL;
 
END_VAR

VAR
	
	color_1_counter                             :UINT;
	color_2_counter                             :UINT;
	orient_1_counter                            :UINT;
	orient_2_counter                            :UINT;
	
	color_cam_1_ok                              :BOOL;
	color_cam_1_nok                             :BOOL;
	color_cam_2_ok                              :BOOL;
	color_cam_2_nok                             :BOOL;
	orient_cam_1_ok                             :BOOL;
	orient_cam_1_nok                            :BOOL;
	orient_cam_2_ok                             :BOOL;
	orient_cam_2_nok                            :BOOL;
	temp_camera_ok                              :BOOL;
END_VAR

VAR
	color1_Toggle_Pos : R_trig;
	color1_Toggle_Neg : F_trig;
	color2_Toggle_Pos : R_trig;
	color2_Toggle_Neg : F_trig;
	orient1_Toggle_Pos : R_trig;
	orient1_Toggle_Neg : F_trig;
	orient2_Toggle_Pos : R_trig;
	orient2_Toggle_Neg : F_trig;
	OP120_color1_seq   : INT;
	OP120_color2_seq   : INT;
	OP120_orient1_seq  : INT;
	OP120_orient2_seq  : INT;
	color1_result_avaliable :BOOL;
	color2_result_avaliable :BOOL;
	orient1_result_avaliable:BOOL;
	orient2_result_avaliable:BOOL;
END_VAR

VAR
////// bypass  button
	
	Lh_color_cam_bypass  :BOOL;
	Lh_orient_cam_bypass :BOOL;
	rh_color_cam_bypass  :BOOL;
    rh_orient_cam_bypass :BOOL;
	
    Lh_color_cam_cmp_bypass: BOOL;
	Lh_orient_cam_cmp_bypass: BOOL;
	rh_color_cam_cmp_bypass: BOOL;
	rh_orient_cam_cmp_bypass: BOOL;
	
	
////// count for color cam
	
	Lh_color_cam_ok_count:LINT;
	Lh_color_cam_nok_count:LINT;
	rh_color_cam_ok_count:LINT;
	rh_color_cam_nok_count:LINT;

////// count for orient cam	

	Lh_orient_cam_ok_count:LINT;
	Lh_orient_cam_nok_count:LINT;
	rh_orient_cam_ok_count:LINT;
	rh_orient_cam_nok_count:LINT;
	
END_VAR

///////////////////////////////       op120 part color camera function block///////////////////////////////////

op120_color_cam_1(
	tTimeout                                                 := , 
	sJob_Name                                                := , 
	camera_ready                                             => op120color1_Camera_Ready,
	Camera_online                                            => op120color1_Camera_Online,
	stCognex_record_status                                   :=op120color1_Acquisition_Status, 
	Acquisition_ID                                           :=op120color1_Acquisition_ID , 
	stCognex_Inspection_status                               :=op120color1_Inspection_Status, 
	Error_Code                                               :=op120color1_Error_code , 
	wcommand_control_in                                      := op120color1_Current_Job_ID, 
	aResults_64_Bytes                                        := op120color1_Cam_Result, 
	number_of_inspections                                    :=op120color1_Inspection_ID , 
	iresult_code                                             := op120color1_Result_code, 
	bTarget_job_ID                                           :=op120color1_Target_Job_ID , 
	Error_Status_message                                     => Error_status, 
	bError                                                   => op120color1_Camera_Error, 
	stCognex_record_control                                  => op120color1_Acquisition_Control , 
	stCognex_inspection_control                              => op120color1_Inspection_Control , 
	wCommandControl_out                                      =>op120color1_Command_word , 
	aUser_data_64_Byte                                       => op120color1_Union.aArrayOfByte, 
	bJob_loading_completed                                   =>op120color1_Job_Change_Complete , 
	bJob_load_failed                                         =>op120color1_Job_Change_Error , 
	bInspection_Result_IO=>  , 
	bInspection_Result_NIO=> , 
	bTXTSM_Error_Job_Change                                  => op120color1_Job_Change_Error, 
	bPictureTakenComplete                                    => op120color1_Picture_Taken, 
	Loaded_Job_ID                                            =>op120color1_Loaded_Job_ID	 , 
	bClear_Error                                             := HMI_Reset, 
	bJob_change_start                                        := op120color1_Camera_Job_Change_start, 
	TXTSM_camera_not_online                                  =>op120color1_Camera_Error	 , 
	bTrigger_start                                           := op120color1_Camera_Trigger );
	
///////////////////////////// op120 color camera 2 function block ////////////////////////////////////////////

op120_color_cam_2(
 tTimeout:= , 
 sJob_Name:= , 
 camera_ready=> op120color2_Camera_Ready,
 Camera_online=> op120color2_Camera_Online,
 stCognex_record_status:=op120color2_Acquisition_Status, 
 Acquisition_ID:=op120color2_Acquisition_ID , 
 stCognex_Inspection_status:=op120color2_Inspection_Status, 
 Error_Code:=op120color2_Error_code , 
 wcommand_control_in:= op120color2_Current_Job_ID, 
 aResults_64_Bytes:= op120color2_Cam_Result, 
 number_of_inspections:=op120color2_Inspection_ID , 
 iresult_code:= op120color2_Result_code, 
 bTarget_job_ID:=op120color2_Target_Job_ID , 
 Error_Status_message=> Error_status, 
 bError=> op120color2_Camera_Error, 
 stCognex_record_control=>op120color2_Acquisition_Control , 
 stCognex_inspection_control=>op120color2_Inspection_Control , 
 wCommandControl_out=>op120color2_Command_word , 
 aUser_data_64_Byte=> op120color2_Union.aArrayOfByte, 
 bJob_loading_completed=>op120color2_Job_Change_Complete , 
 bJob_load_failed=>op120color2_Job_Change_Error , 
 bInspection_Result_IO=>  , 
 bInspection_Result_NIO=> , 
 bTXTSM_Error_Job_Change=> op120color2_Job_Change_Error, 
 bPictureTakenComplete=> op120color2_Picture_Taken, 
 Loaded_Job_ID=>op120color2_Loaded_Job_ID  , 
 bClear_Error:= HMI_Reset, 
 bJob_change_start:= op120color2_Camera_Job_Change_start, 
 TXTSM_camera_not_online=>op120color2_Camera_Error  , 
 bTrigger_start:= op120color2_Camera_Trigger );
 
/////////////////////////       op120 part orientation camera function block///////////////////////////////////	

op120_orient_cam_1(
	tTimeout:= , 
	sJob_Name:= , 
	camera_ready=> op120orient1_Camera_Ready,
	Camera_online=> op120orient1_Camera_Online,
	stCognex_record_status:=op120orient1_Acquisition_Status, 
	Acquisition_ID:=op120orient1_Acquisition_ID , 
	stCognex_Inspection_status:=op120orient1_Inspection_Status, 
	Error_Code:=op120orient1_Error_code , 
	wcommand_control_in:= op120orient1_Current_Job_ID, 
	aResults_64_Bytes:= op120orient1_Cam_Result, 
	number_of_inspections:=op120orient1_Inspection_ID , 
	iresult_code:= op120orient1_Result_code, 
	bTarget_job_ID:=op120orient1_Target_Job_ID , 
	Error_Status_message=> Error_status, 
	bError=> op120orient1_Camera_Error, 
	stCognex_record_control=>op120orient1_Acquisition_Control , 
	stCognex_inspection_control=>op120orient1_Inspection_Control , 
	wCommandControl_out=>op120orient1_Command_word , 
	aUser_data_64_Byte=> op120orient1_Union.aArrayOfByte, 
	bJob_loading_completed=>op120orient1_Job_Change_Complete , 
	bJob_load_failed=>op120orient1_Job_Change_Error , 
	bInspection_Result_IO=>  , 
	bInspection_Result_NIO=> , 
	bTXTSM_Error_Job_Change=> op120orient1_Job_Change_Error, 
	bPictureTakenComplete=> op120orient1_Picture_Taken, 
	Loaded_Job_ID=>op120orient1_Loaded_Job_ID	 , 
	bClear_Error:= HMI_Reset, 
	bJob_change_start:= op120orient1_Camera_Job_Change_start, 
	TXTSM_camera_not_online=>op120orient1_Camera_Error	 , 
	bTrigger_start:= op120orient1_Camera_Trigger );
	
	/////////////////////////////////// op120 orientation camera 2 function block //////////////////////////////
	
 op120_orient_cam_2(
 tTimeout:= , 
 sJob_Name:= , 
 camera_ready=> op120orient2_Camera_Ready,
 Camera_online=> op120orient2_Camera_Online,
 stCognex_record_status:=op120orient2_Acquisition_Status, 
 Acquisition_ID:=op120orient2_Acquisition_ID , 
 stCognex_Inspection_status:=op120orient2_Inspection_Status, 
 Error_Code:=op120orient2_Error_code , 
 wcommand_control_in:= op120orient2_Current_Job_ID, 
 aResults_64_Bytes:= op120orient2_Cam_Result, 
 number_of_inspections:=op120orient2_Inspection_ID , 
 iresult_code:= op120orient2_Result_code, 
 bTarget_job_ID:=op120orient2_Target_Job_ID , 
 Error_Status_message=> Error_status, 
 bError=> op120orient2_Camera_Error, 
 stCognex_record_control=>op120orient2_Acquisition_Control , 
 stCognex_inspection_control=>op120orient2_Inspection_Control , 
 wCommandControl_out=>op120orient2_Command_word , 
 aUser_data_64_Byte=> op120orient2_Union.aArrayOfByte, 
 bJob_loading_completed=>op120orient2_Job_Change_Complete , 
 bJob_load_failed=>op120orient2_Job_Change_Error , 
 bInspection_Result_IO=>  , 
 bInspection_Result_NIO=> , 
 bTXTSM_Error_Job_Change=> op120orient2_Job_Change_Error, 
 bPictureTakenComplete=> op120orient2_Picture_Taken, 
 Loaded_Job_ID=>op120orient2_Loaded_Job_ID  , 
 bClear_Error:= HMI_Reset, 
 bJob_change_start:= op120orient2_Camera_Job_Change_start, 
 TXTSM_camera_not_online=>op120orient2_Camera_Error  , 
 bTrigger_start:= op120orient2_Camera_Trigger );
	
/////////////////////////////// op120 set user data /////////////////////////////////////////////////////////////////////////

IF op120_modelselected = 1 THEN
   op120orient2_Union.aArrayOfByte[0] :=1;
   op120orient1_Union.aArrayOfByte[0] :=1;	
END_IF

op120orient1_Inspection_Control.Set_User_Data := op120_setuserdata;
op120orient2_Inspection_Control.Set_User_Data := op120_setuserdata;

IF op120orient1_Inspection_Status.Set_User_Data_Ack AND op120orient2_Inspection_Status.Set_User_Data_Ack THEN
	op120_setuserdata :=FALSE;
END_IF

////////////////////////////// all camera status //////////////////////////////////
IF (((op120color1_Camera_Ready AND op120color1_Camera_Online) OR Lh_color_cam_bypass OR Lh_color_cam_cmp_bypass )AND
   ((op120color2_Camera_Ready AND op120color2_Camera_Online) OR rh_color_cam_bypass OR rh_color_cam_cmp_bypass) AND
   (( op120orient1_Camera_Ready AND op120orient1_Camera_Online ) OR Lh_orient_cam_bypass OR Lh_orient_cam_cmp_bypass )AND
   (( op120orient2_Camera_Ready AND op120orient2_Camera_Online ) OR rh_orient_cam_bypass OR rh_orient_cam_cmp_bypass )) THEN                                                                                                    
	op120_all_camera_ok := TRUE;	
ELSE op120_all_camera_ok := FALSE;																								 
END_IF		  



	
///////////////////	////////// op 120 camera sequence //////////////////////////////////////////////////////////////////////
 
op120color1_Camera_Trigger:=NOT Lh_color_cam_cmp_bypass AND  OP120_Camera_Auto_Trigger ;
op120orient1_Camera_Trigger:= NOT Lh_orient_cam_cmp_bypass AND OP120_Camera_Auto_Trigger ;
op120color2_Camera_Trigger:= NOT rh_color_cam_cmp_bypass AND OP120_Camera_Auto_Trigger ;
op120orient2_Camera_Trigger:= NOT rh_orient_cam_cmp_bypass AND OP120_Camera_Auto_Trigger ;


//////////////////////////////// toggle bits ////////////////////////////////////////////////////


color1_Toggle_Pos(CLK:=op120color1_Inspection_Status.Inspection_Completed);
color1_Toggle_Neg(CLK:=op120color1_Inspection_Status.Inspection_Completed);
color2_Toggle_Pos(CLK:=op120color2_Inspection_Status.Inspection_Completed);
color2_Toggle_Neg(CLK:=op120color2_Inspection_Status.Inspection_Completed);
orient1_Toggle_Pos(CLK:=op120orient1_Inspection_Status.Inspection_Completed);
orient1_Toggle_Pos(CLK:=op120orient1_Inspection_Status.Inspection_Completed);
orient2_Toggle_Pos(CLK:=op120orient2_Inspection_Status.Inspection_Completed);
orient2_Toggle_Pos(CLK:=op120orient2_Inspection_Status.Inspection_Completed);


////////////////////////////////////////////// camera sequence///////////////////////////////////////////////

CASE  OP120_color1_seq OF
	0: IF op120_auto AND  OP120_Camera_Auto_Trigger THEN
		   OP120_color1_seq               := 10;
	END_IF
	
	10: IF color1_Toggle_Pos.q OR  color1_Toggle_Neg.q THEN
		   IF (op120color1_Cam_Result[0]=1 AND op120color1_Cam_Result[0]<>0) OR temp_camera_ok  
               OR Lh_color_cam_bypass OR Lh_color_cam_cmp_bypass  THEN
	          color_cam_1_ok              := TRUE;
	          color_cam_1_nok             := FALSE;
			     IF NOT  lh_color_cam_bypass THEN
			     Lh_color_cam_ok_count       := Lh_color_cam_ok_count+1;
			     END_IF
			  color1_result_avaliable     := TRUE;
	          OP120_color1_seq            := 0;
            ELSIF NOT Lh_color_cam_bypass AND op120color1_Cam_Result[0]=0 AND op120color1_Cam_Result[0]<>1 THEN
	              color_cam_1_ok          := FALSE;
	              color_cam_1_nok         := TRUE;
				  IF NOT  lh_color_cam_bypass THEN
				  Lh_color_cam_nok_count       := Lh_color_cam_nok_count+1;
				  END_IF
				  color1_result_avaliable := TRUE;
				  OP120_color1_seq        := 0;
             END_IF
	END_IF
END_CASE


CASE  OP120_color2_seq OF
	0: IF op120_auto AND  OP120_Camera_Auto_Trigger THEN
		   OP120_color2_seq                :=10;
	END_IF
	
	10: IF color2_Toggle_Pos.q OR  color2_Toggle_Neg.q THEN
		   IF (op120color2_Cam_Result[0]=1 AND op120color2_Cam_Result[0]<>0) OR temp_camera_ok 
               OR rh_color_cam_bypass OR rh_color_cam_cmp_bypass THEN
	          color_cam_2_ok               := TRUE;
	          color_cam_2_nok              := FALSE;
			    IF NOT rh_color_cam_bypass THEN
			    rh_color_cam_ok_count        :=rh_color_cam_ok_count+1;
			    END_IF
			  color2_result_avaliable      :=TRUE;
	          OP120_color2_seq             := 0;
            ELSIF NOT rh_color_cam_bypass AND op120color2_Cam_Result[0]=0 AND op120color2_Cam_Result[0]<>1 THEN
	              color_cam_2_ok           := FALSE;
	              color_cam_2_nok          := TRUE;
				  IF NOT rh_color_cam_bypass THEN
				  rh_color_cam_nok_count   :=rh_color_cam_nok_count+1;
				  END_IF
				  color2_result_avaliable:=TRUE;
				  OP120_color2_seq         := 0;
             END_IF
	END_IF
END_CASE

CASE  OP120_orient1_seq OF
	0: IF op120_auto AND  OP120_Camera_Auto_Trigger THEN
		   OP120_orient1_seq               := 10;
	END_IF
	
	10: IF color2_Toggle_Pos.q OR  color2_Toggle_Neg.q THEN
		   IF (op120orient1_Cam_Result[1]=1 AND op120orient1_Cam_Result[2]=0) OR temp_camera_ok 
              OR Lh_orient_cam_bypass OR Lh_orient_cam_cmp_bypass THEN
	          orient_cam_1_ok              := TRUE;
	          orient_cam_1_nok             :=FALSE;
			  IF NOT Lh_orient_cam_bypass THEN
			  Lh_orient_cam_ok_count:=Lh_orient_cam_ok_count+1;	  
			  END_IF
			  orient1_result_avaliable     :=TRUE;
	          OP120_orient1_seq            := 0;
            ELSIF NOT Lh_orient_cam_bypass AND  op120orient1_Cam_Result[1]=0 AND op120orient1_Cam_Result[2]=1 THEN
	              orient_cam_1_ok          := FALSE;
	              orient_cam_1_nok         :=TRUE;
				  IF NOT Lh_orient_cam_bypass THEN
				  Lh_orient_cam_nok_count:=Lh_orient_cam_nok_count+1;	  
				  END_IF
				  orient1_result_avaliable :=TRUE;
				  OP120_orient1_seq        := 0;
             END_IF
	END_IF
END_CASE

CASE  OP120_orient2_seq OF
	0: IF op120_auto AND  OP120_Camera_Auto_Trigger THEN
		   OP120_orient2_seq               := 10;
	END_IF
	
	10: IF color2_Toggle_Pos.q OR  color2_Toggle_Neg.q THEN
		   IF (op120orient2_Cam_Result[1]=1 AND op120orient2_Cam_Result[2]=0) OR temp_camera_ok 
               OR rh_orient_cam_bypass OR rh_orient_cam_cmp_bypass THEN
	           orient_cam_2_ok             := TRUE;
	           orient_cam_2_nok            :=FALSE;
			   IF NOT rh_orient_cam_bypass THEN
			   rh_orient_cam_ok_count:=rh_orient_cam_ok_count+1;	   
			   END_IF
			   orient2_result_avaliable    :=TRUE;
	           OP120_orient2_seq := 0;
            ELSIF NOT rh_orient_cam_bypass AND  op120orient2_Cam_Result[1]=0 AND op120orient2_Cam_Result[2]=1 THEN
	              orient_cam_2_ok          := FALSE;
	              orient_cam_2_nok         :=TRUE;
				  IF  NOT rh_orient_cam_bypass THEN
				  rh_orient_cam_nok_count:=rh_orient_cam_nok_count+1;	  
				  END_IF
				  orient2_result_avaliable :=TRUE;
				  OP120_orient2_seq        := 0;
             END_IF
	END_IF
END_CASE


/////////////////////////////////////// op120 camera results ///////////////////////////////////////////////////////////////////

IF orient2_result_avaliable AND orient1_result_avaliable AND color2_result_avaliable AND color1_result_avaliable THEN
IF (color_cam_1_ok AND color_cam_2_ok AND orient_cam_1_ok AND orient_cam_2_ok ) THEN
   OP120_CamOK                              :=TRUE;
   OP120_CamNOK                             :=FALSE;
   color_cam_1_ok                           :=FALSE;
   color_cam_2_ok                           :=false;
   orient_cam_1_ok                          :=false;
   orient_cam_2_ok                          :=false;
   color_cam_1_nok                          :=false;
   color_cam_2_nok                          :=false;
   orient_cam_1_nok                         :=false;
   orient_cam_2_nok                         :=FALSE;
   orient2_result_avaliable                 :=FALSE;
   orient1_result_avaliable                 :=FALSE;
   color2_result_avaliable                  :=FALSE;
   color1_result_avaliable                  :=FALSE;
   
ELSIF  ( color_cam_1_nok OR color_cam_2_nok OR orient_cam_1_nok OR orient_cam_2_nok ) THEN
        OP120_CamOK                         :=FALSE;
        OP120_CamNOK                        :=TRUE;
		color_cam_1_ok                      :=FALSE;
		color_cam_2_ok                      :=FALSE;
		orient_cam_1_ok                     :=FALSE;
		orient_cam_2_ok                     :=FALSE;
		color_cam_1_nok                     :=FALSE;
		color_cam_2_nok                     :=FALSE;
		orient_cam_1_nok                    :=FALSE;
		orient_cam_2_nok                    :=FALSE;
        orient2_result_avaliable            :=FALSE;
        orient1_result_avaliable            :=FALSE;
        color2_result_avaliable             :=FALSE;
	    color1_result_avaliable             :=FALSE;
		
END_IF
END_IF





// color camera 1 result
(*IF (op120color1_Cam_Result[0]=1 AND op120color1_Cam_Result[0]<>0 AND color_1_counter <> op120color1_Inspection_ID)OR temp_camera_ok  THEN
	          color_cam_1_ok := TRUE;
	          color_cam_1_nok:= FALSE;
	          color_1_counter:=op120color1_Inspection_ID;
            ELSIF op120color1_Cam_Result[0]=0 AND op120color1_Cam_Result[0]<>1 AND color_1_counter <> op120color1_Inspection_ID THEN
	              color_cam_1_ok := FALSE;
	              color_cam_1_nok:= TRUE;
             END_IF


// color camera 2 result

IF (op120color2_Cam_Result[0]=1 AND   op120color2_Cam_Result[0]<>0 AND color_2_counter <> op120color2_Inspection_ID) OR temp_camera_ok THEN
	color_cam_2_ok := TRUE;
	color_cam_2_nok:= FALSE;
	color_2_counter:=op120color2_Inspection_ID;

ELSIF op120color2_Cam_Result[0]=0 AND op120color2_Cam_Result[0] <> 1 AND color_2_counter <> op120color2_Inspection_ID THEN
	  color_cam_2_ok := FALSE;
	  color_cam_2_nok:= TRUE;
END_IF

// orient camera 1 result

IF (op120orient1_Cam_Result[1]=1 AND op120orient1_Cam_Result[2]=0 AND orient_1_counter <> op120orient1_Inspection_ID) OR temp_camera_ok THEN
	orient_cam_1_ok := TRUE;
	orient_cam_1_nok:=FALSE;
	orient_1_counter := op120orient1_Inspection_ID;
	
ELSIF op120orient1_Cam_Result[1]=0 AND op120orient1_Cam_Result[2]=1 AND orient_1_counter <> op120orient1_Inspection_ID THEN
	  	orient_cam_1_ok := FALSE;
	    orient_cam_1_nok:=TRUE;
END_IF

// orient camera 2 result

IF (op120orient2_Cam_Result[1]=1 AND op120orient2_Cam_Result[2]=0 AND orient_2_counter <> op120orient2_Inspection_ID) OR temp_camera_ok THEN
	orient_cam_2_ok := TRUE;
	orient_cam_2_nok:=FALSE;
	orient_2_counter := op120orient2_Inspection_ID;
ELSIF op120orient2_Cam_Result[1]=0 AND op120orient2_Cam_Result[2]=1 AND orient_2_counter <> op120orient2_Inspection_ID THEN
	  	orient_cam_2_ok := FALSE;
	    orient_cam_2_nok:=TRUE;
END_IF *)

END_PROGRAM

// ---- POUs/Programs/OP120/OP120_Manual.TcPOU
PROGRAM OP120_Manual
VAR
	
	OP120Enable: BOOL;
	Op120bhome: BOOL;
	op120bset: BOOL;
	temp : bool;
	vel_temp: LREAL;
	Op120_Robot: FB_Robot;
	
	OP120_Robo_Automanual_out: BOOL;
	temp5                    : BOOL;
	temp6                    : BOOL;
	temp7                    : BOOL;
	
END_VAR

///////////////////////////////////////////////Lifting Cylinder function block////////////////////////////////////////////

//move ZERO to STATUS
OP120_Lifting_Cyl_Status:=0;

//Reset Auto Cmd IN Manual Mode & Homing
IF ( OP120_HomeRunning) THEN
	CR120_Lifting_Cyl.AutoCmd1:=FALSE;
	CR120_Lifting_Cyl.AutoCmd2:=FALSE;		
END_IF

// Safe Home
IF (TRUE) AND  (TRUE) THEN 
	CR120_Lifting_Cyl.SafeHome:= TRUE ;
	ELSE 
		CR120_Lifting_Cyl.SafeHome:= FALSE ;
	END_IF
// Safe Work
IF (TRUE) OR (TRUE) THEN 
	CR120_Lifting_Cyl.Safework:= TRUE ;
	ELSE 
		CR120_Lifting_Cyl.Safework:= FALSE ;
	END_IF
	
// Manual PB  Cyl Mapping
IF (CR120_HMI_Lifting_Cyl_Home_PB=TRUE) THEN
	CR120_Lifting_Cyl.ManualPB1:=TRUE;
	ELSE 
		CR120_Lifting_Cyl.ManualPB1:=FALSE;
	END_IF
	
IF (CR120_HMI_Lifting_Cyl_Work_PB=TRUE) THEN
	CR120_Lifting_Cyl.ManualPB2:=TRUE;
	ELSE 
		CR120_Lifting_Cyl.ManualPB2:=FALSE;
	END_IF


	
CR120_Lifting_Cyl(
	Auto:=OP120_AutoSelected , 
	Manual:= OP120_ManualSelected, 
	ErrorActive:=OP120_ErrorActive , 
	ResetPB:=OP120_HMI_Reset , 
	Sensor1:=I120_LH_SING_CYL_REV_I1220_2 , 
	Sensor2:=I120_LH_SING_CYL_FWD_I1220_3 , 
	ManualPB1:= , 
	ManualPB2:= , 
	AutoCmd1:= , 
	AutoCmd2:= , 
	OperationEnable:=OperationEnable , 
	SafeHome:= , 
	SafeWork:= , 
	HomingCmd1:= , 
	Pulse_1Sec:=Pulse_Block.Q1Hz , 
	BlinkingBit:= , 
	TimeOut1:=5 , 
	TimeOut2:=5 , 
	TimeOut3:=5 , 
	Solenoid1=>O120_LH_SING_CYL_REV_Q1261_4 , 
	Solenoid2=>O120_LH_SING_CYL_FWD_Q1261_5 , 
	AlarmSensor1=>berror[1119] , 
	AlarmSensor2=>berror[1120] , 
	AlarmSolenoid1=>berror[1121] , 
	AlarmSolenoid2=>berror[1122] , 
	AllSignal=>berror[1123] , 
	AlarmPresent=> , 
	Position1=> , 
	Position2=> , 
	HomeSensorBlink=> , 
	WorkSensorBlink=> , 
	Status:=OP120_Lifting_Cyl_Status );
	
/////////////////////////////////////////////gripper cylinder function block///////////////////////////////////////

//move ZERO to STATUS
OP120_Gripper_Cyl_Status:=0;



//Reset Auto Cmd IN Manual Mode & Homing
IF (OP120_Auto OR OP120_HomeRunning) THEN
	CR120_Gripper_Cyl.AutoCmd1:=FALSE;
	CR120_Gripper_Cyl.AutoCmd2:=FALSE;		
END_IF

// Safe Home
IF (TRUE) AND  (TRUE) THEN 
	CR120_Gripper_Cyl.SafeHome:= TRUE ;
	ELSE 
		CR120_Gripper_Cyl.SafeHome:= FALSE ;
	END_IF
// Safe Work
IF (TRUE) OR (TRUE) THEN 
	CR120_Gripper_Cyl.Safework:= TRUE ;
	ELSE 
		CR120_Gripper_Cyl.Safework:= FALSE ;
	END_IF
	
// Manual PB  Cyl Mapping
IF (CR120_HMI_Gripper_Cyl_Home_PB=TRUE) THEN
	CR120_Gripper_Cyl.ManualPB1:=TRUE;
	ELSE 
		CR120_Gripper_Cyl.ManualPB1:=FALSE;
	END_IF
	
IF (CR120_HMI_Gripper_Cyl_Work_PB=TRUE) THEN
	CR120_Gripper_Cyl.ManualPB2:=TRUE;
	ELSE 
		CR120_Gripper_Cyl.ManualPB2:=FALSE;
	END_IF


	
CR120_Gripper_Cyl(
	Auto:=OP120_AutoSelected , 
	Manual:= OP120_ManualSelected, 
	ErrorActive:=OP120_ErrorActive , 
	ResetPB:=OP120_HMI_Reset , 
	Sensor1:= NOT (I120_LH_LOCKSPRING_GRPR_CLSE_I405_4 OR I120_RH_LOCKSPRING_GRPR_CLSE_I405_6)  , 
	Sensor2:=(I120_LH_LOCKSPRING_GRPR_CLSE_I405_4 OR I120_RH_LOCKSPRING_GRPR_CLSE_I405_6), 
	ManualPB1:= , 
	ManualPB2:= , 
	AutoCmd1:=OP120_EO_RO_Gripper1_Open , 
	AutoCmd2:=OP120_EO_RO_Gripper1_Close , 
	OperationEnable:=OperationEnable , 
	SafeHome:= , 
	SafeWork:= , 
	HomingCmd1:= , 
	Pulse_1Sec:=Pulse_Block.Q1Hz , 
	BlinkingBit:= , 
	TimeOut1:=50 , 
	TimeOut2:=50 , 
	TimeOut3:=50 , 
	Solenoid1=>O120_LH_GRPR_OPN_Q1260_5 , 
	Solenoid2=>O120_LH_GRPR_CLSE_Q1260_4 , 
	AlarmSensor1=>berror[1104], 
	AlarmSensor2=>berror[1105] , 
	AlarmSolenoid1=>berror[1106] , 
	AlarmSolenoid2=>berror[1107] , 
	AllSignal=>berror[1108] , 
	AlarmPresent=> , 
	Position1=> temp7 , 
	Position2=>   temp6, 
	HomeSensorBlink=> , 
	WorkSensorBlink=> , 
	Status:=OP120_Gripper_Cyl_Status );
	
	IF temp7 THEN
		OP120_EI_Gripper1_Open:=TRUE;
		OP120_EI_Gripper2_Open:=TRUE;
		ELSE
			OP120_EI_Gripper1_Open:=FALSE;
		OP120_EI_Gripper2_Open:=FALSE;
		END_IF
	IF temp6 THEN
		OP120_EI_Gripper1_Close:=TRUE;
		OP120_EI_Gripper2_Close:=TRUE;
		ELSE
			OP120_EI_Gripper1_Close:=FALSE;
		OP120_EI_Gripper2_Close:=FALSE;
		END_IF
///////////////////////////////////////////////// Horizontal Push Cyl function block////////////////////////////////////

//move ZERO to STATUS
OP120_Horizontal_Push_Cyl_Status:=0;



//Reset Auto Cmd IN Manual Mode & Homing
IF  (OP120_HomeRunning) THEN
	CR120_Horizontal_Push_Cyl.AutoCmd1:=FALSE;
	CR120_Horizontal_Push_Cyl.AutoCmd2:=FALSE;		
END_IF

// Safe Home
IF (TRUE) AND  (TRUE) THEN 
	CR120_Horizontal_Push_Cyl.SafeHome:= TRUE ;
	ELSE 
		CR120_Horizontal_Push_Cyl.SafeHome:= FALSE ;
	END_IF
// Safe Work
IF (TRUE) OR (TRUE) THEN 
	CR120_Horizontal_Push_Cyl.Safework:= TRUE ;
	ELSE 
	CR120_Horizontal_Push_Cyl.Safework:= FALSE ;
	END_IF

// Manual PB  Cyl Mapping
IF (CR120_HMI_Horizontal_Push_Cyl_Home_PB=TRUE) THEN
	CR120_Horizontal_Push_Cyl.ManualPB1:=TRUE;
	ELSE 
		CR120_Horizontal_Push_Cyl.ManualPB1:=FALSE;
	END_IF
	
IF (CR120_HMI_Horizontal_Push_Cyl_Work_PB=TRUE) THEN
	CR120_Horizontal_Push_Cyl.ManualPB2:=TRUE;
	ELSE 
		CR120_Horizontal_Push_Cyl.ManualPB2:=FALSE;
	END_IF

CR120_Horizontal_Push_Cyl(
	Auto:=OP120_AutoSelected , 
	Manual:=OP120_ManualSelected , 
	ErrorActive:= OP120_ErrorActive, 
	ResetPB:=OP120_HMI_Reset , 
	Sensor1:= I120_PUSH_CYL_REV_I1220_0, 
	Sensor2:=I120_PUSH_CYL_FWD_I1220_1 , 
	ManualPB1:= , 
	ManualPB2:= , 
	AutoCmd1:= , 
	AutoCmd2:= , 
	OperationEnable:= OperationEnable, 
	SafeHome:= , 
	SafeWork:= , 
	HomingCmd1:= , 
	Pulse_1Sec:= Pulse_Block.Q1Hz, 
	BlinkingBit:= , 
	TimeOut1:= 5, 
	TimeOut2:=5 , 
	TimeOut3:=5 , 
	Solenoid1=>O120_PUSH_CYL_REV_Q1261_2 , 
	Solenoid2=>O120_PUSH_CYL_FWD_Q1261_3 , 
	AlarmSensor1=>berror[1114] , 
	AlarmSensor2=>berror[1115] , 
	AlarmSolenoid1=>berror[1116] , 
	AlarmSolenoid2=>berror[1117] , 
	AllSignal=>berror[1118] , 
	AlarmPresent=> , 
	Position1=> , 
	Position2=> , 
	HomeSensorBlink=> , 
	WorkSensorBlink=> , 
	Status:=OP120_Horizontal_Push_Cyl_Status );
	
	// Camera Slide Cylinder
	
	

//move ZERO to STATUS
OP120_Camera_Slide_Cyl_Status:=0;



//Reset Auto Cmd IN Manual Mode & Homing
IF (OP120_Auto OR OP120_HomeRunning) THEN
	CR120_Camera_Slide_Cyl.AutoCmd1:=FALSE;
	CR120_Camera_Slide_Cyl.AutoCmd2:=FALSE;		
END_IF

// Safe Home
IF (TRUE) AND  (TRUE) THEN 
	CR120_Camera_Slide_Cyl.SafeHome:= TRUE ;
	ELSE 
		CR120_Camera_Slide_Cyl.SafeHome:= FALSE ;
	END_IF
// Safe Work
IF (TRUE) OR (TRUE) THEN 
	CR120_Camera_Slide_Cyl.Safework:= TRUE ;
	ELSE 
	CR120_Camera_Slide_Cyl.Safework:= FALSE ;
	END_IF

// Manual PB  Cyl Mapping
IF (CR120_HMI_Camera_Slide_Cyl_Home_PB=TRUE) THEN
	CR120_Camera_Slide_Cyl.ManualPB1:=TRUE;
	ELSE 
		CR120_Camera_Slide_Cyl.ManualPB1:=FALSE;
	END_IF
	
IF (CR120_HMI_Camera_Slide_Cyl_Work_PB=TRUE) THEN
	CR120_Camera_Slide_Cyl.ManualPB2:=TRUE;
	ELSE 
		CR120_Camera_Slide_Cyl.ManualPB2:=FALSE;
	END_IF

CR120_Camera_Slide_Cyl(
	Auto:=OP120_AutoSelected , 
	Manual:=OP120_ManualSelected , 
	ErrorActive:=OP120_ErrorActive , 
	ResetPB:=OP120_HMI_Reset , 
	Sensor1:= I120_CAMERA_SLIDE_CYL_REV_I1220_4, 
	Sensor2:=I120_CAMERA_SLIDE_CYL_FWD_I1220_5 , 
	ManualPB1:= , 
	ManualPB2:= , 
	AutoCmd1:= , 
	AutoCmd2:= , 
	OperationEnable:= OperationEnable, 
	SafeHome:= , 
	SafeWork:= , 
	HomingCmd1:= , 
	Pulse_1Sec:= Pulse_Block.Q1Hz, 
	BlinkingBit:= , 
	TimeOut1:=5 , 
	TimeOut2:= 5, 
	TimeOut3:=5 , 
	Solenoid1=>O120_CAMERA_SLIDECYL_REV_Q1262_0 , 
	Solenoid2=>O120_CAMERA_SLIDECYL_FWD_Q1262_1 , 
	AlarmSensor1=>berror[1109] , 
	AlarmSensor2=>berror[1110] , 
	AlarmSolenoid1=>berror[1111] , 
	AlarmSolenoid2=> berror[1112], 
	AllSignal=>berror[1113] , 
	AlarmPresent=> , 
	Position1=> , 
	Position2=> , 
	HomeSensorBlink=> , 
	WorkSensorBlink=> , 
	Status:=OP120_Camera_Slide_Cyl_Status );
	

	
//////////////////////////////////////////////////Oring feed Servo function block //////////////////////////////////////////////////////////////
	
	
	IF (TRUE) THEN
		SR120_Oring_Feed_Servo_Control.Safety_cond:=TRUE;
	END_IF

vel_temp:= (-50);
	
SR120_Oring_Feed_Servo(
	bAxis1_Ref_Switch:= , 
	bInit:= , 
	bErrorReset:=OP120_HMI_Reset OR Servo_Reset , 
	bEnable:=OperationEnable,
	bMoveVelocity:= , 
	bHalt:= , 
	bManualMode:=OP120_ManualSelected OR OP120Enable , 
	fHomePos:= , 
	fOverride:= , 
	fTargetPosition:= , 
	fTargetVelocity:= SR120_Oring_Feed_Servo_Control.Velocity, 
	fAcc:= , 
	fDec:= , 
	Safe_move_Conditions:=Servo_Safety,
	HME_WRITE_ADD:= 16#5017, 
	Axis:= SR120_Oring_Feed_Servo_Axis, 
	bHome:=Op120bhome, 
	bSetPosition:=op120bset, 
	bMoveVelocity:=SR120_Oring_Feed_Servo_Control.VELmove_Start ,	
	bMoveAbsolute:= SR120_Oring_Feed_Servo_Control.ABSmove_Start, 
	bMoveRelative:=SR120_Oring_Feed_Servo_Control.RELmove_Start , 
	bMoveTorque:=SR120_Oring_Feed_Servo_Control.Torque_mode_Start , 
	stManualModeAxis:=SR120_Oring_Feed_Manual_Axis , 
	bmove_home:=SR120_Oring_Feed_Servo_Control.Axis_Home_Cmd , 
	sAxisState=>SR120_Oring_Feed_Servo_Control.Axis_State , 
	bAxis_ready=>SR120_Oring_Feed_Servo_Control.Axis_ready , 
	bAxisInPosition=>SR120_Oring_Feed_Servo_Control.Axis_In_Pos , 
	bAxisError=>berror[1151]  , 
	bAxisEnabled=>SR120_Oring_Feed_Servo_Control.Axis_Enabled , 
	bAxisHomed=>SR120_Oring_Feed_Servo_Control.Axis_reference , 
	bSetPositionDone=> , 
	bHaltDone=>SR120_Oring_Feed_Servo_Control.Axis_Halted , 
	bSTOPDone=>SR120_Oring_Feed_Servo_Control.Axis_Stopped , 
	bHomeDone=> , 
	bDone=> , 
	bTorqueReached=>SR120_Oring_Feed_Servo_Control.Trq_reached , 
	bsafe_to_move=>SR120_Oring_Feed_Servo_Control.Safety_cond , 
	baxis_in_home_pos=> , 
	bABS_Pos_done=> , 
	Actual_position=> , 
	Actual_velocity=> , 
	Actual_Torque=> );
	
//SR120_Oring_Feed_Manual_Axis.jogPos :=OP120Enable ;	


IF MANUAL_SELECTED AND OP120_ManualSelected THEN               
	IF I120_CONV_REVI600_7 THEN
		SR120_Oring_Feed_Manual_Axis.targetVelocity :=-50.0;
		SR120_Oring_Feed_Manual_Axis.moveVelocity	:=I120_CONV_REVI600_7;
 	ELSIF I120_CONV_FWDI601_0 THEN
		SR120_Oring_Feed_Manual_Axis.targetVelocity :=50.0;
		SR120_Oring_Feed_Manual_Axis.moveVelocity	:=I120_CONV_FWDI601_0;	
	ELSE 	
		SR120_Oring_Feed_Manual_Axis.moveVelocity:=0;   	
	END_IF  	
END_IF
			
//////////////////////////////////////////////////// Robot function block /////////////////////////////////////////////		
				
	Op120_Robot(
	i_b_Operation_Enable_Feedback:= OP120_SO_Auto_Operation_Enable, 
	i_b_Auto_Enable_Feedback:=OP120_SO_Mirror_Auto_enable , 
	i_b_Servo_On_Feedback:= OP120_SO_Servo_ON_OFF_Status, 
	i_b_Servo_Off_Feedback:= OP120_SO_Mirror_SRVO_Off, 
	i_b_Error_Feedback:=OP120_SO_During_error OR OP120_ErrorActive , 
	i_b_Program_Start_Enable_Feedback:=OP120_SO_Program_Execute , 
	i_b_Robo_Stopping_Feedback:=OP120_SO_During_Cycle_Stop , 
	i_b_Emergency_Pressed_Feedback:=OP120_SO_During_EMG_Stop , 
	i_b_Auto_Mode_Feedback:=OP120_SO_Auto_Ext_Mode , 
	i_b_Reset:=OP120_HMI_Reset OR Servo_Reset, 
	i_b_RobotAutoManual:=OP120_Auto AND NOT temp5 , 
	i_b_ProgramReset:=OP120_Robo_ProgramReset , 
	o_b_Operation_Enable_Cmd=>OP120_SI_Operation_Enable , 
	o_b_Auto_Enable_Cmd=>OP120_SI_Auto_Enable , 
	o_b_Servo_On_Cmd=>OP120_SI_Servo_ON , 
	o_b_Servo_Off_Cmd=>OP120_SI_Servo_OFF , 
	o_b_Error_Reset_Cmd=>OP120_SI_Error_Reset , 
	o_b_Program_Reset_Cmd=>OP120_SI_Program_Reset , 
	o_b_Program_Start_Cmd=>OP120_SI_Start , 
	o_b_Program_Stop_Cmd=>OP120_SI_Stop2 , 
	o_b_RobotAutoManual=>OP120_Robo_Automanual_out , 
	o_b_Error=>berror[1150] );

END_PROGRAM

// ---- POUs/Programs/OP120/OP120_Error.TcPOU
PROGRAM OP120_Error
VAR
	OP120_StepErr1:ton;
	OP120_StepErr2:ton;
	OP120_StepErr3:ton;
	bdone: BOOL;
	i: INT;
	Raise: INT;
	j: INT;
	Clear: INT;
END_VAR

IF NOT bdone THEN
	bdone:=TRUE;
FOR i:=1100 TO 1200 BY 1 DO 
	
IF berror[i] THEN
	OP120_ErrorActive:=TRUE;
END_IF
END_FOR
bdone:=FALSE;
END_IF

IF OP120_HMI_Reset OR Servo_Reset THEN
	FOR j:=1100 TO 1200 BY 1 DO 
		
	
	berror[j]:=FALSE;
	OP120_ErrorActive:=FALSE;
	
	END_FOR
	temp:=false;
END_IF

END_PROGRAM

// ---- POUs/Programs/OP120/OP120_Initialization_Seq.TcPOU
PROGRAM OP120_Initialization_Seq
VAR
	Op120_temphomeTrig: R_TRIG;
	TempHome: BOOL;
	ROboProgResetDly: TON;
	Master_reset :BOOL;
	robot_homed : BOOL;
	op120_Home_seq_done   :BOOL;
	op120_model_selected  :INT;
	air_purge_off         :ton;
	air_purge_on          :BOOL;
END_VAR

IF NOT OP120_HomeRunning AND OP120_GVL.CR120_Lifting_Cyl.Position1 AND  OP120_GVL.CR120_Horizontal_Push_Cyl.Position1 AND ( OP120_IO_Tag_link.OP120_SO_Rbt_In_Home OR robot_homed )THEN
	OP120_GVL.OP120_Temp_Home_OK:=TRUE;
	OP120_HomeRunning:=FALSE;
	OP120_Homing_Seq:=0;
	TempHome:=FALSE;
	air_purge_on      :=FALSE;
ELSE
	OP120_GVL.OP120_Temp_Home_OK:=FALSE;
END_IF

// reset bits set during error active
IF   OP120_GVL.OP120_AutoRunning OR  OP120_GVL.OP120_StepRunning OR OP120_ErrorActive THEN
	 op120_Home_seq_done :=FALSE;
     robot_homed := FALSE;
END_IF

CASE OP120_Homing_Seq OF
	
	0: IF (OP120_Auto AND NOT OP120_HomeRunning AND  NOT OP120_ErrorActive AND  NOT OP120_GVL.OP120_AutoRunning AND NOT OP120_GVL.OP120_StepRunning	AND NOT op120_Home_seq_done) THEN
		OP120_HomeRunning:=TRUE;
		OP120_Homing_Seq:=5;	
	   END_IF
	   
	  5:IF (OP120_HomeRunning AND OP120_GVL.OP120_HMI_Homing_PB )THEN
		  // OP120_GVL.OP120_Vaccuum_OP_Port5_Byte1 :=1;
	      // OP120_GVL.OP120_Vaccuum_OP_Port6_Byte1 :=1;
           O120_LH_REJ_AIR_PURGE_Q1261_6 :=TRUE;
	       O120_SPARE_Q1262_3:=TRUE;
           air_purge_on      :=TRUE; 
           IF NOT OP120_Vaccum1_Bit0 AND NOT OP120_Vaccum2_Bit0 AND air_purge_off.q THEN  
              O120_LH_REJ_AIR_PURGE_Q1261_6 :=FALSE;
		      O120_SPARE_Q1262_3:=FALSE;
              air_purge_on      :=FALSE;            
              OP120_Homing_Seq:=10;
        END_IF
		END_IF
		
	 10:  IF (OP120_HomeRunning )THEN  
		      OP120_GVL.CR120_Horizontal_Push_Cyl.HomingCmd1:= TRUE;
			  OP120_GVL.CR120_Lifting_Cyl.HomingCmd1:= TRUE;
			  IF OP120_GVL.CR120_Horizontal_Push_Cyl.Position1 AND OP120_GVL.CR120_Lifting_Cyl.Position1  THEN
			     OP120_GVL.CR120_Horizontal_Push_Cyl.HomingCmd1:= FALSE;
			     OP120_GVL.CR120_Lifting_Cyl.HomingCmd1:= FALSE;
			     OP120_Homing_Seq:=20;
			  END_IF
	      END_IF
		  
		
  
	20:	  IF (OP120_HomeRunning)THEN
		      OP120_Robo_ProgramReset:=TRUE;
	          IF ROboProgResetDly.Q AND NOT OP120_SO_Program_Execute THEN
		         OP120_Robo_ProgramReset:=FALSE;
		         OP120_Homing_Seq:=30;
	           END_IF
	       END_IF
		   
	30:  IF (OP120_HomeRunning)AND NOT Master_reset THEN
		     OP120_Robo_Out6001:=1;//3
			 OP120_SI_Homing_Start:=TRUE;
			 OP120_Homing_Seq:=40;
		 ELSIF (OP120_HomeRunning)AND  Master_reset THEN
			    OP120_Robo_Out6001:=3;//1
			    OP120_SI_Homing_Start:=TRUE;
				OP120_Homing_Seq:=40;
	     END_IF
		 
	40:  IF (OP120_HomeRunning)AND OP120_SO_Rbt_In_Home THEN
		     OP120_SI_Homing_Start:=FALSE;
			 robot_homed := TRUE;
			 OP120_Homing_Seq:=50;
	    END_IF
	
    50:	IF (OP120_HomeRunning) AND robot_homed THEN
            op120_Home_seq_done :=TRUE;
		    OP120_HomeRunning:=FALSE;
            OP120_Homing_Seq:=60; 
		END_IF	
		
	60:	IF op120_all_camera_ok THEN
		   op120_setuserdata:=TRUE;
           OP120_Homing_Seq:=0;
		END_IF  
			
END_CASE

IF NOT OP120_HomeRunning THEN
	OP120_GVL.CR120_Horizontal_Push_Cyl.HomingCmd1:= FALSE;
	OP120_GVL.CR120_Lifting_Cyl.HomingCmd1:= FALSE;
END_IF

Op120_temphomeTrig(CLK:=TempHome , Q=> );
ROboProgResetDly(IN:= OP120_Robo_ProgramReset, PT:= T#200MS, Q=> , ET=> );
air_purge_off(IN:=air_purge_on , PT:=T#500MS, Q=> , ET=> );

END_PROGRAM

// ---- POUs/Programs/OP120/OP120_AutoSequence.TcPOU
PROGRAM OP120_AutoSequence
VAR
	OP120_AutoSeq:INT;
	OP120_Moverinstationtrig: R_TRIG;
	continuousrunplsdelete: BOOL;
	dry_run: BOOL;
	fix_lh: INT;
	fix_rh: INT;
	op120_cycle_time_fb :FB_cycleTime;
	OP120_Cycle_time : UDINT;
	OP120_ROBO_ERR   :TON;
	
END_VAR

VAR PERSISTENT
	OP120_ROBO_ERR_TIME: TIME;
END_VAR

IF (NOT OP120_Auto OR  OP120_ErrorActive OR OP120_HomeRunning OR OP120_Machine_Stop ) THEN
	OP120_GVL.OP120_AutoRunning:= FALSE;
	OP120_ComponentOk:=FALSE;
	OP120_ComponentNok:=FALSE;
	OP120_OperationCompleted:=FALSE;
	OP120_PushPlace:=FALSE;
	Part_Picked:=FALSE;
	Ready_for_next_singulation:=FALSE;
	OP120_AutoSeq:= 10;
	OP120_MoverPresent:=FALSE;
    Op120_PartSingulated:=FALSE;
	OP120_GVL.OP120_Vaccuum_OP_Port5_Byte1 :=1;
	OP120_GVL.OP120_Vaccuum_OP_Port6_Byte1 :=1;
END_IF


OP120_ROBO_ERR(IN:=	NOT(OP120_SO_Auto_Operation_Enable AND OP120_SO_Mirror_Auto_enable AND OP120_SO_Servo_ON_OFF_Status) , PT:=OP120_ROBO_ERR_TIME, Q=> , ET=> );


CASE OP120_AutoSeq OF 
	10:IF (OP120_Auto) THEN		// Check Automode Selected
		OP120_AutoSeq :=20;
	    END_IF
	20:IF ( NOT OP120_ErrorActive) THEN		//Check No error
		OP120_AutoSeq:=30;
	   END_IF
	30:IF (NOT OP120_HomeRunning) THEN		//Check No Homerunning
		OP120_AutoSeq :=40;
		END_IF
    40:IF ( OP120_GVL.OP120_Temp_Home_OK)THEN	//Check Machine in Home
		OP120_AutoSeq:= 50;
		END_IF
	50:IF ( NOT OP120_OperationCompleted) THEN		// Check Operation Completed Reset
		OP120_AutoSeq:=60;
		END_IF
	60:IF (NOT OP120_ComponentOk) THEN		// Check Component Ok Reset
		OP120_AutoSeq:=70;
		END_IF
	70:IF (NOT OP120_ComponentNok) THEN 	// Check Component NOk Reset
		   OP120_AutoSeq:= 120;
		END_IF
		
    120:IF  (AUTO_RUNNING OR (NOT AUTO_RUNNING AND OP120_GVL.OP120_HMI_CycleStart_PB )) THEN		//Machine Start in Fully Automatic or Press Cycle Start For Semi Automatic
		    OP120_GVL.OP120_HomeCondition_OK:=TRUE;
	 			IF( OP120_GVL.OP120_HomeCondition_OK AND OP120_AutoSelected) THEN
					OP120_GVL.OP120_AutoRunning:=TRUE;
					OP120_GVL.OP120_StepRunning:= FALSE;
				
				ELSIF (OP120_Main.OP120_Modeselection_FB.HomeConditionOK AND OP120_StepSelected) THEN
					OP120_GVL.OP120_AutoRunning:=FALSE;
					OP120_GVL.OP120_StepRunning:= TRUE;
				END_IF;
		 END_IF
		 IF ((OP120_GVL.OP120_AutoRunning OR OP120_GVL.OP120_StepRunning) AND OP120_GVL.OP120_StartEnable) THEN
			OP120_Prev_Comp_Status:=1;
		    OP120_Sing_AutoSeq:=10;
		    OP120_AutoSeq:= 140;
		END_IF
		
		
	140: IF OP120_STN_ENABLE AND fix_lh <> 110 AND fix_rh <> 110 THEN   //// waiting for station enable and previous component status
         	OP120_AutoSeq:= 200;
			
         ELSIF OP120_STN_ENABLE AND fix_lh =110 AND fix_rh =110 THEN
           OP120_Prev_LH_COMP_OK:=TRUE;
	       OP120_Prev_RH_COMP_OK:=TRUE;
           OP120_Prev_LH_COMP_NOK:=FALSE;
           OP120_Prev_RH_COMP_NOK:=FALSE;
		  
         ELSIF OP120_STN_ENABLE AND fix_lh = 110 AND fix_rh =111 THEN
           OP120_Prev_LH_COMP_OK:=TRUE;
	       OP120_Prev_RH_COMP_OK:=FALSE;
           OP120_Prev_LH_COMP_NOK:=FALSE;
           OP120_Prev_RH_COMP_NOK:=TRUE;
		   
         ELSIF OP120_STN_ENABLE AND fix_lh = 111 AND fix_rh =110 THEN
           OP120_Prev_LH_COMP_OK:=FALSE;
	       OP120_Prev_RH_COMP_OK:=TRUE;
		   OP120_Prev_LH_COMP_NOK:=TRUE;
           OP120_Prev_RH_COMP_NOK:=FALSE;
          END_IF 
		  
          IF (OP120_Prev_LH_COMP_OK OR OP120_Prev_LH_COMP_NOK) AND (OP120_Prev_RH_COMP_OK OR OP120_Prev_RH_COMP_NOK) THEN
			 
			  OP120_Lock_AutoSeq:=10;
			  
	          OP120_AutoSeq:= 150;
		  END_IF	
  
	150:	IF OP120_StartEnable AND OP120_STN_ENABLE OR continuousrunplsdelete THEN /// waiting for station enable
			IF continuousrunplsdelete THEN
	           OP120_STN_ENABLE := TRUE;
	        END_IF
            OP120_MoverPresent:=TRUE;
			OP120_AutoSeq:= 160;
			END_IF
	
	160:	IF OP120_StartEnable THEN
		       OP120_AutoSeq:= 170;
        	END_IF
			
170:     IF OP120_OperationCompleted  AND (OP120_STN_MOVER>0 OR dry_run) THEN // waiting for operation complete feedback
	     	IF OP120_LH_Comp_OK AND OP120_rH_Comp_OK THEN
	     		MOVER_CMP_STATUS[OP120_CURR_MOVER][1]:=120;	
                 MOVER_CMP_STATUS[OP120_CURR_MOVER][2]:=120;
	     	    IF MOVER_CMP_STATUS[OP120_CURR_MOVER][1]=120 AND MOVER_CMP_STATUS[OP120_CURR_MOVER][2]=120 AND MOVER_CMP_STATUS[OP120_STN_MOVER][1] <> 110 AND MOVER_CMP_STATUS[OP120_STN_MOVER][2]<>110 THEN
	     		STATION_DONE[OP120_CURR_MOVER][OP120_XTS_POS_NO]			:= TRUE;
				   IF continuousrunplsdelete THEN
	                  OP120_STN_ENABLE := FALSE;
	               END_IF		   
	     		   OP120_AutoSeq:= 250;
				END_IF
	     	 ELSIF OP120_LH_Comp_NOK AND OP120_rH_Comp_OK THEN	
	     		   MOVER_CMP_STATUS[OP120_CURR_MOVER][1]:=121;	
                    MOVER_CMP_STATUS[OP120_CURR_MOVER][2]:=120;
	     	       IF MOVER_CMP_STATUS[OP120_CURR_MOVER][1]=121 AND MOVER_CMP_STATUS[OP120_CURR_MOVER][2]=120 
						AND MOVER_CMP_STATUS[OP120_CURR_MOVER][1] <> 110 AND MOVER_CMP_STATUS[OP120_CURR_MOVER][2]<>110 THEN
	     		    STATION_DONE[OP120_CURR_MOVER][OP120_XTS_POS_NO]			:= TRUE;
	     		      OP120_AutoSeq:= 250;
	     		    END_IF
               ELSIF OP120_LH_Comp_OK AND OP120_rH_Comp_NOK THEN	
	     			MOVER_CMP_STATUS[OP120_CURR_MOVER][1]:=120;	
                     MOVER_CMP_STATUS[OP120_CURR_MOVER][2]:=121;
	     	        IF MOVER_CMP_STATUS[OP120_CURR_MOVER][1]=120 AND MOVER_CMP_STATUS[OP120_CURR_MOVER][2]=121 
						AND MOVER_CMP_STATUS[OP120_CURR_MOVER][1] <> 110 AND MOVER_CMP_STATUS[OP120_CURR_MOVER][2]<>110 THEN
	     		    STATION_DONE[OP120_CURR_MOVER][OP120_XTS_POS_NO]			:= TRUE;
	     		       OP120_AutoSeq:= 250;
	     		     END_IF	
	     	  ELSIF OP120_LH_Comp_NOK AND OP120_rH_Comp_NOK THEN	
	     		    MOVER_CMP_STATUS[OP120_CURR_MOVER][1]:=121;	
                     MOVER_CMP_STATUS[OP120_CURR_MOVER][2]:=121;
	     	        IF MOVER_CMP_STATUS[OP120_CURR_MOVER][1]=121 AND MOVER_CMP_STATUS[OP120_CURR_MOVER][2]=121 
						AND MOVER_CMP_STATUS[OP120_CURR_MOVER][1] <> 110 AND MOVER_CMP_STATUS[OP120_CURR_MOVER][2]<>110 THEN
	     		  STATION_DONE[OP120_CURR_MOVER][OP120_XTS_POS_NO]			:= TRUE;
	     		       OP120_AutoSeq:= 250;
                      END_IF
	             END_IF
	     END_IF

	200:MOVER_CMP_STATUS[OP120_CURR_MOVER][1]:=121;	
        MOVER_CMP_STATUS[OP120_CURR_MOVER][2]:=121;
		IF MOVER_CMP_STATUS[OP120_CURR_MOVER][1]=121 AND MOVER_CMP_STATUS[OP120_CURR_MOVER][2]=121 
			AND MOVER_CMP_STATUS[OP120_CURR_MOVER][1] <> 110 AND MOVER_CMP_STATUS[OP120_CURR_MOVER][2]<>110 THEN
		STATION_DONE[OP120_CURR_MOVER][OP120_XTS_POS_NO]			:= TRUE;
			OP120_AutoSeq:= 250;
		END_IF
		
	250:// Reset All Bits							
//        IF NOT OP120_STN_ENABLE THEN         reseting all bits for next cycle
		 OP120_LH_Comp_OK:=FALSE;
         OP120_LH_Comp_NOK:=FALSE;
         OP120_RH_Comp_OK:=FALSE;
         OP120_RH_Comp_NOK:=FALSE;
         OP120_LH_AutoSeq:=0;
		 OP120_RH_AutoSeq:=0;
		 OP120_OperationCompleted:=FALSE;
		 OP120_AutoSeq:= 140;
//		END_IF
END_CASE

OP120_Moverinstationtrig(CLK:= OP120_MoverinStation, Q=> );
op120_cycle_time_fb(i_b_startTime:=OP120_STN_ENABLE , i_b_stopTime:= NOT OP120_STN_ENABLE , o_t_StationTime=>OP120_Cycle_time );

dry_run:=All_Station_Dry_Run;
//staus FOR movers 
IF  dry_run THEN
	fix_lh :=110;
	fix_rh :=110;
ELSE 
	fix_lh := MOVER_CMP_STATUS[OP120_STN_MOVER][1];
	fix_rh := MOVER_CMP_STATUS[OP120_STN_MOVER][2];
END_IF


//############################		OP120 STATION ENABLE CONDITION		##########################

	OP120_STN_MOVER					:= MOVER_POSITION[OP120_XTS_POS_NO];
	IF AUTO_WITH_XTS THEN
	IF OP120_STN_MOVER>0  AND NOT OP120_STN_ENABLE THEN		
	IF NOT(END_OF_CYCLE AND MOVER_CMP_STATUS[OP120_STN_MOVER][1]=5 AND MOVER_CMP_STATUS[OP120_STN_MOVER][2]=5)THEN
	OP120_STN_ENABLE					:= MOVER_POS_RECHED[OP120_STN_MOVER] AND ((MOVER_CMP_STATUS[OP120_STN_MOVER][1]=110)OR 
										(MOVER_CMP_STATUS[OP120_STN_MOVER][2]=110))AND STATION_ENABLE_CONTROL;
	ELSE
		STATION_DONE[OP120_STN_MOVER][OP120_XTS_POS_NO]			:= TRUE;		
	END_IF
	ELSE
	OP120_STN_ENABLE					:= FALSE;
	END_IF
	END_IF

END_PROGRAM

// ---- POUs/Programs/OP120/OP120_Feed_Conveyor.TcPOU
PROGRAM OP120_Feed_Conveyor
VAR	
	conveyor_forward         :BOOL;
	conveyor_reverse         :BOOL;
	rev_time                 :INT;
    feed_conveyor_seq        :INT;
	bowl_over_flow           :BOOL;
	bowl_filled              :BOOL;
	bowl_on_off_tmr          :ton;
	hopper_off_tme           :ton;
	air_purge_1              :ton;
	air_purge_2              :ton;
	reverse_run_time         :ton;
END_VAR

VAR PERSISTENT
	frd_speed:LREAL;
	rev_speed:LREAL;
END_VAR

(*
IF (NOT OP120_GVL.OP120_AutoSelected OR OP120_GVL.OP120_ErrorActive) THEN
	OP120_GVL.OP120_AutoRunning:= FALSE;
	OP120_GVL.SR130_Oring_Feed_Servo_Control.VELmove_Start:=FALSE;
	forward:=FALSE;
	reverse:=FALSE;
	con_step_no:= 10;
END_IF	*)
IF (NOT OP120_Auto OR  OP120_ErrorActive OR OP120_HomeRunning OR OP120_Machine_Stop ) THEN
	feed_conveyor_seq:=0;
END_IF

CASE feed_conveyor_seq OF
	

		0: IF (OP120_GVL.OP120_AutoSelected) THEN		// Check Automode Selected
				feed_conveyor_seq:=20;
				conveyor_status  := 1;    ///////////// waiting for auto selection
	        END_IF
		
	    20:IF (NOT OP120_GVL.OP120_ErrorActive) THEN		//Check No error
		       feed_conveyor_seq:=60;
			   conveyor_status  := 2;    /////////////// waiting for error reset
      	   END_IF
	
		   
		60:IF (  OP120_AutoRunning  ) AND NOT Op120_PartSingulated  THEN		//Machine Start in Fully Automatic or Press Cycle Start For Semi Automatic
				OP120_GVL.OP120_Vaccuum_OP_Port5_Byte1 :=0;
		        OP120_GVL.OP120_Vaccuum_OP_Port6_Byte1 :=0;
               feed_conveyor_seq:= 65;	
			    conveyor_status  := 3;  /////////// turning on vaccum
		   END_IF
		   
		65: IF  NOT  (OP120_Vaccum1_Bit0 AND OP120_Vaccum2_Bit0) THEN
   				 feed_conveyor_seq:= 70;
				 conveyor_status  := 4;  /////////// component not present in singulation unit
			ELSE
				 feed_conveyor_seq:= 90;
				 conveyor_status  := 5;  /////////// component present in the singulation unit
			END_IF
     
			
		70: 	OP120_GVL.SR120_Oring_Feed_Servo_Control.Velocity:= frd_speed;
				SR120_Oring_Feed_Servo.bHalt:=FALSE;				
				conveyor_forward:=TRUE;
    	    	OP120_GVL.SR120_Oring_Feed_Servo_Control.VELmove_Start:=TRUE;
		         conveyor_status  := 6; ////// conveyor moving forward and waiting for vaccum feedback
				IF OP120_Vaccum1_Bit0 AND OP120_Vaccum2_Bit0 THEN
					
					 OP120_GVL.SR120_Oring_Feed_Servo_Control.VELmove_Start:=FALSE;
					 SR120_Oring_Feed_Servo.bHalt:=TRUE;
					 
					 IF SR120_Oring_Feed_Servo_Control.Axis_Halted THEN
						OP120_GVL.SR120_Oring_Feed_Servo_Control.VELmove_Start:=FALSE;
						SR120_Oring_Feed_Servo.bHalt:=FALSE;
						conveyor_forward:=FALSE;	
					    feed_conveyor_seq:= 90;
					END_IF
				END_IF
				
		
		90: 	OP120_GVL.SR120_Oring_Feed_Servo_Control.Velocity:=rev_speed;
				SR120_Oring_Feed_Servo.bHalt:=FALSE;
				conveyor_reverse:=TRUE;
				conveyor_status  := 8; ////  conveyor moving reverse to singulate the part
				OP120_GVL.SR120_Oring_Feed_Servo_Control.VELmove_Start:=TRUE;
				IF reverse_run_time.Q THEN
					OP120_GVL.SR120_Oring_Feed_Servo_Control.VELmove_Start:=FALSE;
					SR120_Oring_Feed_Servo.bHalt:=TRUE;
					IF SR120_Oring_Feed_Servo_Control.Axis_Halted THEN
						SR120_Oring_Feed_Servo.bHalt:=FALSE;
						Op120_PartSingulated:=TRUE;
						conveyor_reverse:=FALSE;
						feed_conveyor_seq:= 60;
						conveyor_status  := 9;  // PART singulated TO the fixture
					END_IF
				END_IF				
END_CASE

///////// timer for feed conveyor
reverse_run_time(IN:= conveyor_reverse, PT:= INT_TO_TIME(100), Q=> , ET=> );



/////////////////////////////////////////////////hopper and bowl logic//////////////////////////////////////////////////////////////////	
	
    //Bowl  Control through selector switch in manual mode 
	IF NOT OP120_HMI_AutoMode AND OP120_HMI_ManualMOde AND NOT OP120_HMI_StepMode AND NOT OP120_Gvl.OP120_ErrorActive  THEN
	       O120_BOWL_ENABLEQ600_1:=I120_BOWL_OFF_ONI600_5 OR Op120_Gvl.OP120_HMI_Bowl_On_PB;
	END_IF 
	
	IF (I120_BOWL_OFF_ONI600_5 AND Op120_Gvl.OP120_HMI_Bowl_On_PB) OR OP120_Gvl.OP120_ErrorActive THEN
		O120_BOWL_ENABLEQ600_1:= FALSE;
	END_IF
	
	// bowl auto logic
	IF (OP120_Gvl.OP120_AutoSelected) THEN
	   Op120_Gvl.OP120_HMI_Bowl_On_PB:=FALSE;
	END_IF
	
	IF  (OP120_HMI_AutoMode OR OP120_HMI_StepMode) AND NOT OP120_HMI_ManualMOde   AND NOT OP120_Gvl.OP120_ErrorActive  AND NOT bowl_on_off_tmr.Q THEN
		 O120_BOWL_ENABLEQ600_1:= TRUE;
		                        
	ELSIF (OP120_HMI_AutoMode OR OP120_HMI_StepMode) AND NOT OP120_HMI_ManualMOde   AND NOT OP120_Gvl.OP120_ErrorActive AND bowl_on_off_tmr.Q THEN	
           O120_BOWL_ENABLEQ600_1:= FALSE;
	END_IF

	bowl_over_flow := I120_VBF_CONV_TRK2_OVERFLWI601_2 AND I120_VBF_CONV_TRK1_OVERFLW_I601_1 AND OP120_HMI_AutoMode ;
	bowl_on_off_tmr(IN:= bowl_over_flow, PT:=T#2S, Q=> , ET=> );
	
	//hopper Control through selector switch in manual mode 
	
	IF NOT OP120_HMI_AutoMode AND OP120_HMI_ManualMOde AND NOT OP120_HMI_StepMode AND NOT OP120_Gvl.OP120_ErrorActive AND (I120_HPR_OFF_ONI600_6 OR Op120_Gvl.OP120_HMI_Hopper_On_PB ) THEN   //AND I120_BOWL_LOW_LVLI600_4
	   O120_HPR_ENABLEQ600_0 :=FALSE;
	 END_IF   
	 
	 IF NOT OP120_HMI_AutoMode AND OP120_HMI_ManualMOde AND NOT OP120_HMI_StepMode AND (NOT I120_HPR_OFF_ONI600_6 AND NOT Op120_Gvl.OP120_HMI_Hopper_On_PB )OR OP120_Gvl.OP120_ErrorActive THEN
	     O120_HPR_ENABLEQ600_0:= TRUE;
	 END_IF	 
	 
	//hopper auto logic
	
	IF (OP120_Gvl.OP120_AutoSelected) THEN
	  Op120_Gvl.OP120_HMI_Hopper_On_PB:=FALSE;
	END_IF
	 
	 IF (OP120_HMI_AutoMode OR OP120_HMI_StepMode) AND NOT OP120_HMI_ManualMOde   AND NOT OP120_Gvl.OP120_ErrorActive AND NOT I120_BOWL_LOW_LVLI600_4 THEN 
	    O120_HPR_ENABLEQ600_0:=FALSE;
	 ELSIF hopper_off_tme.Q THEN
		 O120_HPR_ENABLEQ600_0:=TRUE;
	 END_IF	
	 
	bowl_filled := I120_BOWL_LOW_LVLI600_4 ;
	hopper_off_tme(IN:= bowl_filled AND (OP120_HMI_AutoMode OR OP120_HMI_StepMode) AND NOT OP120_HMI_ManualMOde, PT:= T#1S, Q=> , ET=> );
	
//////// air purge auto sequence/////////
	
IF  air_purge_2.Q AND NOT OP120_Gvl.OP120_ErrorActive AND (OP120_HMI_AutoMode OR OP120_HMI_StepMode) AND NOT OP120_HMI_ManualMOde THEN
	O120_SPARE_Q1262_5 := TRUE;
	ELSE 
    O120_SPARE_Q1262_5 := FALSE;	
END_IF
	
IF  Air_purge_1.Q AND NOT OP120_Gvl.OP120_ErrorActive AND (OP120_HMI_AutoMode OR OP120_HMI_StepMode) AND NOT OP120_HMI_ManualMOde THEN
	O120_SPARE_Q1262_4 := TRUE;
	ELSE 
	O120_SPARE_Q1262_4 := FALSE;	
END_IF
	
/// timer for bowl feeder air purge ///	

air_purge_1(IN:= I120_VBF_CONV_TRK1_OVERFLW_I601_1 AND NOT I120_VBF_CONV_TRK2_OVERFLWI601_2 , PT:= T#2S, Q=> , ET=> );
air_purge_2(IN:=I120_VBF_CONV_TRK2_OVERFLWI601_2 AND NOT I120_VBF_CONV_TRK1_OVERFLW_I601_1 , PT:=T#2S , Q=> , ET=> );

//// bowl tower lamp logic

IF OP120_AutoSelected AND (O120_BOWL_ENABLEQ600_1 OR NOT O120_HPR_ENABLEQ600_0) THEN
   O120_HPR_TWR_LMP_GREENQ600_3	 := Pulse_Block.Q0_5Hz;
ELSIF NOT OP120_AutoSelected  AND (O120_BOWL_ENABLEQ600_1 OR NOT O120_HPR_ENABLEQ600_0) THEN
	O120_HPR_TWR_LMP_REDQ600_2   :=  Pulse_Block.Q5Hz ;
END_IF

END_PROGRAM

// ---- POUs/Programs/OP120/OP120_LockInsert_AutoSequence.TcPOU
PROGRAM OP120_LockInsert_AutoSequence
VAR
	operation :INT;
	Pushing_Dly: TON;
	PushDly: TON;
	PullDly:TON;
	OP120_MoverDly: TON;
	
END_VAR

IF NOT OP120_StartEnable THEN
	OP120_Lock_AutoSeq:=0;
END_IF
CASE OP120_Lock_AutoSeq OF 
	
	10:IF OP120_StartEnable THEN
		OP120_Lock_AutoSeq:=20;
	END_IF
	
	20:IF OP120_StartEnable AND CheckParkOK AND NOT OP120_EO_Spring_Pick_Completed THEN
		OP120_GotoPick:=TRUE;
		OP120_Lock_AutoSeq:=30;
		robot_status :=1; ///// waiting for ready to pick command
		ELSIF OP120_StartEnable AND OP120_EO_Spring_Pick_Completed THEN
		OP120_Lock_AutoSeq:=35;	
	END_IF
	
	30:IF OP120_StartEnable AND OP120_EO_Spring_Pick_Completed   THEN
		  Part_Picked:=TRUE;
		  Ready_for_next_singulation:=TRUE;
		  OP120_GotoPick:=FALSE;
		  OP120_Lock_AutoSeq:=35;
		  robot_status :=2; // part picked and waiting for place ommmand
		ELSIF OP120_StartEnable AND NOT  OP120_EO_Spring_Pick_Completed   THEN
			robot_status :=3; /// waiting for part pick feedback
	   END_IF
	
	35:IF OP120_StartEnable  THEN
		OP120_Lock_AutoSeq:=36;
	END_IF
	
	36: IF OP120_StartEnable AND OP120_MoverPresent THEN
		   OP120_Lock_AutoSeq:=40;
		ELSIF  OP120_StartEnable AND OP120_MoverPresent THEN
           robot_status :=4; /// waiting for mover present feedback 
	    END_IF
	
	40:IF OP120_StartEnable AND OP120_EO_Spring_Place_Pos_Reached THEN
		OP120_PushPlace:=TRUE;
		Part_Picked:=FALSE;
		OP120_MoverPresent:=FALSE;
		OP120_Lock_AutoSeq:=50;
		ELSIF  OP120_StartEnable AND NOT  OP120_EO_Spring_Place_Pos_Reached THEN
			     robot_status :=5; /// waiting for place pos reach feedback
		
	END_IF
	
	50:IF OP120_StartEnable AND OP120_PushPlace   THEN
		CR120_Horizontal_Push_Cyl.AutoCmd2:=TRUE;
		CR120_Horizontal_Push_Cyl.AutoCmd1:=FALSE;
		IF CR120_Horizontal_Push_Cyl.Position2 AND PushDly.Q THEN
		OP120_Lock_AutoSeq:=60;
		ELSIF NOT  CR120_Horizontal_Push_Cyl.Position2 THEN
			  robot_status :=6; /// waiting lock spring insert cyl work feedback
	    END_IF
	     
	     END_IF
		OP120_CURR_MOVER			:=OP120_STN_MOVER;
	
	60:IF OP120_StartEnable THEN
		CR120_Horizontal_Push_Cyl.AutoCmd1:=TRUE;
		CR120_Horizontal_Push_Cyl.AutoCmd2:=FALSE;
		IF CR120_Horizontal_Push_Cyl.Position1 AND PullDly.Q THEN
			OP120_LH_Comp_OK:=TRUE;
	        OP120_rH_Comp_OK:=TRUE;
		    OP120_Lock_AutoSeq:=70;
		    OP120_PartPushed:=TRUE;
		ELSIF NOT CR120_Horizontal_Push_Cyl.Position1 THEN	
			robot_status :=7; /// waiting lock spring insert cyl home feedback
	    END_IF
	    END_IF
	
	70:IF OP120_StartEnable AND OP120_EO_Spring_Place_Completed THEN
		OP120_PushPlace:=FALSE;
		OP120_PartPushed:=FALSE;
		Op120_PartPlaced:=TRUE;
		OP120_Lock_AutoSeq:=80;
		ELSIF NOT OP120_EO_Spring_Place_Completed THEN
			  robot_status :=8; /// waiting for plae complete feedback from robot 
		END_IF
		
	80: IF OP120_StartEnable AND NOT OP120_EO_Spring_Place_Completed AND OP120_MoverDly.q THEN
		
		Op120_PartPlaced:=FALSE;
		OP120_Lock_AutoSeq:=81;
		OP120_OperationCompleted:=TRUE;
		operation:=operation+1;
	    END_IF
	
	81 :IF  OP120_OperationCompleted THEN
		  //  OP120_Lock_AutoSeq:=10;
	END_IF
	
 
END_CASE

PushDly(IN:=(OP120_Lock_AutoSeq=50 AND CR120_Horizontal_Push_Cyl.Position2 )  , PT:=T#0S , Q=> , ET=> );
PullDly(IN:=(OP120_Lock_AutoSeq=60 AND CR120_Horizontal_Push_Cyl.Position1 )  , PT:=T#0S , Q=> , ET=> );


OP120_MoverDly(IN:=(OP120_Lock_AutoSeq=80) , PT:=T#0.2S , Q=> , ET=> );

END_PROGRAM

// ---- POUs/Programs/OP120/OP120_Sing_Auto_PRG.TcPOU
PROGRAM OP120_Sing_Auto_PRG
VAR	
	next_singulation:BOOL;
	next_singulation_time:ton;
	singulation_down     :TON;
	cam_nok_count     :INT;
	purge_delay       :ton;
	purge_on          :BOOL;
	cyl_delay         :BOOL;
	cyl_down          :ton;
	time_1            :INT;
	time_2            :int;
END_VAR

IF NOT OP120_StartEnable THEN
	
	OP120_Sing_AutoSeq        :=0;
	OP120_Camera_Auto_Trigger := FALSE;
	CheckParkNOK              := FALSE;
	CheckParkOK               := FALSE;
	OP120_CamOK               := FALSE;
	OP120_CamNOK              := FALSE;
	cam_nok_count             :=0;
	 purge_on                 := false;
	
END_IF

CASE   OP120_Sing_AutoSeq OF 
	
	10:IF OP120_GVL.OP120_StartEnable AND  Op120_PartSingulated   THEN    
          CR120_Lifting_Cyl.AutoCmd2:=TRUE;
		  CR120_Lifting_Cyl.AutoCmd1:=FALSE;
		  IF CR120_Lifting_Cyl.Position2 THEN
		     OP120_Sing_AutoSeq:= 160;
		  ELSIF NOT CR120_Lifting_Cyl.Position2 THEN
                conveyor_status  := 11; /// waiting for singulation cylinder work feedback	 
	      END_IF
		ELSIF NOT  Op120_PartSingulated THEN
               conveyor_status  := 10;   // waiting for part singulated feedback
	    END_IF
		
	160:IF OP120_GVL.OP120_StartEnable AND NOT  OP120_SO_Rbt_In_Pick_Zone THEN      // enabling camera for part check
		   OP120_Camera_Auto_Trigger:=TRUE;
		   OP120_Sing_AutoSeq:= 170;	
         ELSIF  OP120_SO_Rbt_In_Pick_Zone THEN 
                conveyor_status  := 12; // waiting for robot not in pick zone feedback
	    END_IF
		
	170: IF OP120_GVL.OP120_StartEnable THEN      // waiting for camera feedback
           IF OP120_CamOK  THEN  
		       CheckParkOK:=TRUE;
		       CheckParkNOK:=FALSE;
		       OP120_Camera_Auto_Trigger:=FALSE;
		       OP120_Sing_AutoSeq:= 180;
		   
		    END_IF
			
		   IF OP120_CamNOK  THEN
			  OP120_Camera_Auto_Trigger:=FALSE;
			  cam_nok_count := cam_nok_count+1;
			  OP120_Sing_AutoSeq:= 190;
			  CheckParkNOK:=TRUE;
			  CheckParkOK:=FALSE;
			 
			END_IF	 
		 ELSIF 	OP120_GVL.OP120_StartEnable AND NOT OP120_CamOK AND NOT OP120_CamNOK THEN
			     conveyor_status  := 13; // waiting for camera result
		END_IF

	180: IF OP120_StartEnable AND (Ready_for_next_singulation OR singulation_down.q) THEN  //PartPickedTrig.q	     
		     CheckParkNOK:=FALSE;
			 CheckParkOK:=FALSE;
			 next_singulation:=TRUE;
			 Ready_for_next_singulation:=FALSE;
			 OP120_Sing_AutoSeq:= 181;
			 conveyor_status  := 14; 
		 ELSIF 	 OP120_StartEnable AND NOT Ready_for_next_singulation THEN
			     conveyor_status  := 14; // camera result ok waiting for robot to pick
		END_IF	 
		
	181 : IF OP120_StartEnable AND 	next_singulation_time.Q AND NOT (OP120_Vaccum1_Bit0 AND OP120_Vaccum2_Bit0) THEN 
		      next_singulation:=0;
			  Op120_PartSingulated:=FALSE;
			  OP120_Sing_AutoSeq:= 200;
			ELSIF NOT  OP120_Vaccum1_Bit0 AND OP120_Vaccum2_Bit0 THEN
                  conveyor_status  := 15; ////  waiting for vacum feedback cutoff after robot pick
		  END_IF	 
	         
	190: IF OP120_StartEnable AND CheckParkNOK THEN
		    OP120_GVL.OP120_Vaccuum_OP_Port5_Byte1 :=1;
			OP120_GVL.OP120_Vaccuum_OP_Port6_Byte1 :=1;
			purge_on := TRUE;
			conveyor_status  := 16; ////  camera nok and purge is turned on
		IF purge_delay.Q THEN
               O120_LH_REJ_AIR_PURGE_Q1261_6 :=TRUE;
		       O120_SPARE_Q1262_3:=TRUE;
			  
		IF  NOT OP120_Vaccum1_Bit0 AND NOT OP120_Vaccum2_Bit0 THEN
		           OP120_GVL.OP120_Vaccuum_OP_Port5_Byte1 :=0;
			       OP120_GVL.OP120_Vaccuum_OP_Port6_Byte1 :=0;
                   O120_LH_REJ_AIR_PURGE_Q1261_6 :=FALSE;
		           O120_SPARE_Q1262_3:=FALSE;
		           Op120_PartSingulated:=FALSE;
				   purge_on := FALSE;
				   cyl_delay :=TRUE;
		           OP120_Sing_AutoSeq:= 200;
		ELSIF  OP120_Vaccum1_Bit0 OR OP120_Vaccum2_Bit0  THEN
					conveyor_status  := 17; ////  waiting for vacum cut off 
		END_IF  
	    END_IF
        END_IF
		  
	200: IF OP120_StartEnable AND cyl_down.Q   THEN	
	        OP120_CamOK:=FALSE;
	        OP120_CamNOK:=FALSE;   
		    CheckParkNOK:=FALSE;
			CheckParkOK := FALSE;
		    CR120_Lifting_Cyl.AutoCmd1:=TRUE;
		    CR120_Lifting_Cyl.AutoCmd2:=FALSE;
			conveyor_status  := 18; /// waitng singulation cylinder home
		  IF CR120_Lifting_Cyl.Position1 THEN
		     OP120_Sing_AutoSeq:= 10;
		 END_IF
		 END_IF
		 
END_CASE



// ton

next_singulation_time(IN:=  next_singulation, PT:=T#0MS , Q=> , ET=> );
purge_delay(IN:=purge_on , PT:= INT_TO_TIME(time_1), Q=> , ET=> );
cyl_down(IN:= cyl_delay, PT:=INT_TO_TIME(time_2) , Q=> , ET=> );
singulation_down(IN:= OP120_Sing_AutoSeq=180 AND ( NOT OP120_Vaccum1_Bit0 OR NOT OP120_Vaccum2_Bit0) , PT:=T#500MS , Q=> , ET=> );

END_PROGRAM

// ---- POUs/Programs/OP130/OP130_Main.TcPOU
PROGRAM OP130_Main
VAR
	OP130_Modeselection_FB: Mode_Selection_Block1;
	
	
	
	
	Times: LREAL;
	Start: BOOL;
	// Servo Offline Testings
	LH_Cylinder_Offline_FB: cylinder_2_pos;
	RH_Cylinder_Offline_FB: cylinder_2_pos;
	RH_Servo_Offline_Block: servo;
	LH_Servo_Offline_Block: servo;
	RH_Servo_EnableOffline_Block: servo;
	
	Clmap_Servo_Offline_Block: servo;
	OP130_Cycle_Time_FB: FB_cycleTime;
	Error_On: BOOL;
	Error_On_LH: BOOL;
	Error_On_RH: BOOL;
	OP130_Clock: FB_SimClock;
END_VAR

// Function Calling

OP130_Manual();
OP130_AutoSequence();
OP130_LH_Auto();
OP130_RH_Auto();
OP130_Error();
OP130_Initialization_Seq();
OP130_RH_Initialization_Seq();
op130_tool_change();


//MOdeselection From HMI

IF (OP130_HMI_AutoMode AND NOT OP130_HMI_ManualMOde AND NOT OP130_HMI_StepMode) THEN
	OP130_Modeselection_FB.ModeWord:=1;
	ELSIF (NOT OP130_HMI_AutoMode AND OP130_HMI_ManualMOde AND NOT OP130_HMI_StepMode) THEN
		OP130_Modeselection_FB.ModeWord:=2;
	ELSIF  (NOT OP130_HMI_AutoMode AND NOT OP130_HMI_ManualMOde AND  OP130_HMI_StepMode) THEN
		OP130_Modeselection_FB.ModeWord:=3;
    ELSE   
		OP130_Modeselection_FB.ModeWord:=0;
END_IF
	





OP130_Modeselection_FB(
	ModeWord:= , 
	HomeConditionOK:=OP130_Home_ConditionOK , 
	OperationEnable:=OperationEnable , 
	StartPB:=OP130_HMI_Cycle_Start , 
	SafetyAndNOError:=OperationEnable , 
	ModeAck:=TRUE , 
	HomingINProgress:= , 
	TempHomeOK:=OP130_Temp_Home_OK , 
	ResetPB:= , 
	AutoSelected=>OP130_AutoSelected , 
	ManualSelected=>OP130_ManualSelected , 
	StepSelected=>OP130_StepSelected , 
	ModeSelAck_Indication=> , 
	StatusDisplay=> , 
	AutoRunning:=OP130_AutoRunning , 
	StepRunning:=OP130_StepRunning , 
	StartEnable:=OP130_StartEnable , 
	MachineStop:=OP130_Machine_Stop );
	
	
	IF OP130_AutoSelected OR OP130_StepSelected THEN
		OP130_Auto:=TRUE;
		ELSE
			OP130_Auto:=FALSE;
		END_IF

END_PROGRAM

// ---- POUs/Programs/offline testing/cylinder_2_pos.TcPOU
FUNCTION_BLOCK cylinder_2_pos
VAR_INPUT
	en_in: BOOL;
	error_bit: BOOL;
	cylinder_work_coil:BOOL;
	cylinder_home_coil:BOOL;
	delay_1: LTIME;
	delay_2: LTIME;
	
END_VAR
VAR_OUTPUT
	en_out: BOOL;
	cylinder_work_fb:BOOL;
	cylinder_home_fb:BOOL;
	delay_display_1: LTIME;
	delay_display_2: LTIME;
	
END_VAR
VAR
	sensor_delay_1: LTON;
	sensor_delay_2: LTON;
	

	
END_VAR
VAR_IN_OUT
	
END_VAR
VAR // added by the converter: edge detectors and wires of the graphical bodies
    _w1, _w2, _w3 : BOOL;
END_VAR

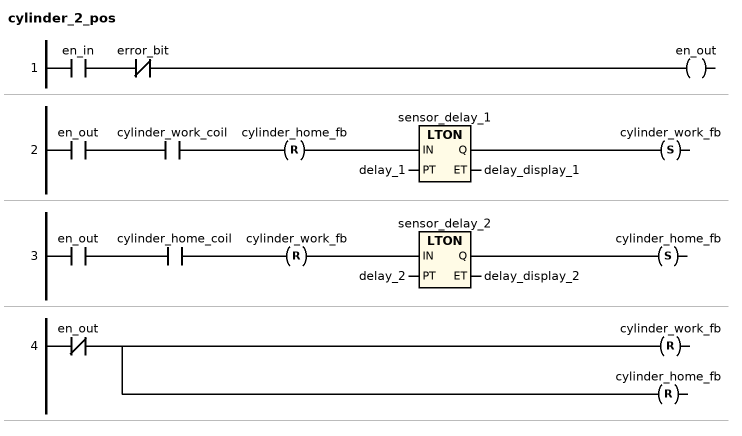
// NETWORK 1
en_out := en_in AND NOT error_bit;

// NETWORK 2
_w1 := en_out AND cylinder_work_coil;
cylinder_home_fb R= _w1;
sensor_delay_1(IN := _w1, PT := delay_1, ET => delay_display_1); // LTON
cylinder_work_fb S= sensor_delay_1.Q;

// NETWORK 3
_w2 := en_out AND cylinder_home_coil;
cylinder_work_fb R= _w2;
sensor_delay_2(IN := _w2, PT := delay_2, ET => delay_display_2); // LTON
cylinder_home_fb S= sensor_delay_2.Q;

// NETWORK 4
_w3 := NOT en_out;
cylinder_work_fb R= _w3;
cylinder_home_fb R= _w3;

END_FUNCTION_BLOCK

// ---- FB/FB_SimClock.TcPOU
FUNCTION_BLOCK FB_SimClock
VAR_INPUT
	
END_VAR
VAR_OUTPUT

Q10Hz				: BOOL;
Q5Hz				: BOOL;
Q2_5Hz				: BOOL;
Q2Hz				: BOOL;
Q1_25Hz				: BOOL;
Q1Hz				: BOOL;
Q0_625Hz			: BOOL;
Q0_5Hz				: BOOL;


END_VAR
VAR
	
T1				: TOF;
T2				: TOF;

R10Hz			: R_Trig;
R5Hz			: R_Trig;
R2_5Hz			: R_Trig;
R2Hz			: R_Trig;
R1_25Hz			: R_Trig;
R1Hz			: R_Trig;
R0_625Hz		: R_Trig;
R0_5Hz			: R_Trig;	
RCTU			: R_Trig;

CTU				: CTU;	
END_VAR

// Clock block with variable pulse width.

T1(IN:=NOT T2.Q , PT:= T#50MS, Q=>Q10Hz , ET=> );
T2(IN:=T1.Q , PT:= T#50MS, Q=> , ET=> );


R10Hz(CLK:=Q10Hz , Q=> );
Q5Hz:= R10Hz.Q XOR Q5Hz;

R5Hz(CLK:=Q5Hz , Q=>);
Q2_5Hz:= R5Hz.Q XOR Q2_5Hz;

R2_5Hz(CLK:=Q2_5Hz , Q=>);
Q1_25Hz:= R2_5Hz.Q XOR Q1_25Hz;

R1_25Hz(CLK:=Q1_25Hz , Q=>);
Q0_625Hz:= R1_25Hz.Q XOR Q0_625Hz;


CTU(
	CU:= Q10Hz, 
	RESET:= ctu.Q, 
	PV:= 5, 
	Q=> , 
	CV=> );
	
	
RCTU(CLK:=ctu.Q , Q=>);	
Q2Hz:= RCTU.Q XOR Q2Hz;
	
	
R2Hz(CLK:=Q2Hz , Q=> );
Q1Hz:= R2Hz.Q XOR Q1Hz;	

R1Hz(CLK:=Q1Hz , Q=> );
Q0_5Hz:= R1Hz.Q XOR Q0_5Hz;

END_FUNCTION_BLOCK

// ---- POUs/Programs/OP130/OP130_Manual.TcPOU
PROGRAM OP130_Manual
VAR

	OP130_Enable: BOOL;
	FESTO_NOT_NEED: BOOL;
	NOT_REQ: BOOL;
	OP130_LH_Servo_Safety: BOOL;
	OP130_RH_Servo_Safety:BOOL;
	CR130_RH_Rotart_Cyl_Stats: INT;
	CR130_LH_Rotart_Cyl_Stats: INT;
END_VAR

//LH Rotary Cylinder

//move ZERO to STATUS
OP130_GVL.CR130_LH_Rotart_Cyl_Status:=0;

//Reset Auto Cmd IN Manual Mode & Homing
IF  (OP130_HomeRunning) THEN
	CR130_LH_Rot_Cyl.AutoCmd1:=FALSE;
	CR130_LH_Rot_Cyl.AutoCmd2:=FALSE;		
END_IF

// Safe Home
IF SR130_stManualModeAxis_LH_Vert_Servo.actualPosition >= 57.0 THEN 
	CR130_LH_Rot_Cyl.SafeHome:= TRUE ;
	ELSE 
		CR130_LH_Rot_Cyl.SafeHome:= FALSE ;
	END_IF
// Safe Work
IF SR130_stManualModeAxis_LH_Vert_Servo.actualPosition >= 57.0 THEN 
	CR130_LH_Rot_Cyl.Safework:= TRUE ;
	ELSE 
		CR130_LH_Rot_Cyl.Safework:= FALSE ;
	END_IF
	
// Manual PB  Cyl Mapping
IF (OP130_HMI_LH_Rotary_Cyl_Home_PB=TRUE) THEN
	CR130_LH_Rot_Cyl.ManualPB1:=TRUE;
	ELSE 
		CR130_LH_Rot_Cyl.ManualPB1:=FALSE;
	END_IF
	
IF (OP130_HMI_LH_Rotary_Cyl_Work_PB=TRUE) THEN
	CR130_LH_Rot_Cyl.ManualPB2:=TRUE;
	ELSE 
		CR130_LH_Rot_Cyl.ManualPB2:=FALSE;
	END_IF


	
